LIN {X 262.840,Y 122.534,Z 110.362,A -155.005,B 90.000,C 0.000} C_DIS
LIN {X 263.458,Y 121.203,Z 110.346,A -155.295,B 90.000,C 0.000} C_DIS
LIN {X 263.907,Y 120.222,Z 110.562,A -155.508,B 90.000,C 0.000} C_DIS
LIN {X 264.680,Y 118.510,Z 111.492,A -155.880,B 90.000,C 0.000} C_DIS
LIN {X 264.694,Y 118.479,Z 111.523,A -155.886,B 90.000,C 0.000} C_DIS
LIN {X 264.792,Y 118.258,Z 111.652,A -155.934,B 90.000,C 0.000} C_DIS
LIN {X 265.375,Y 116.944,Z 112.118,A -156.218,B 90.000,C 0.000} C_DIS
LIN {X 265.872,Y 115.810,Z 112.354,A -156.463,B 90.000,C 0.000} C_DIS
LIN {X 265.934,Y 115.668,Z 112.428,A -156.493,B 90.000,C 0.000} C_DIS
LIN {X 266.916,Y 113.380,Z 112.646,A -156.985,B 90.000,C 0.000} C_DIS
LIN {X 267.884,Y 111.074,Z 112.657,A -157.479,B 90.000,C 0.000} C_DIS
LIN {X 268.826,Y 108.776,Z 112.374,A -157.970,B 90.000,C 0.000} C_DIS
LIN {X 268.883,Y 108.638,Z 112.351,A -158.000,B 90.000,C 0.000} C_DIS
LIN {X 269.020,Y 108.296,Z 112.339,A -158.072,B 90.000,C 0.000} C_DIS
LIN {X 268.155,Y 110.420,Z 113.333,A -157.619,B 90.000,C 0.000} C_DIS
LIN {X 267.237,Y 112.623,Z 114.079,A -157.148,B 90.000,C 0.000} C_DIS
LIN {X 266.268,Y 114.897,Z 114.450,A -156.659,B 90.000,C 0.000} C_DIS
LIN {X 266.207,Y 115.038,Z 114.463,A -156.629,B 90.000,C 0.000} C_DIS
LIN {X 265.209,Y 117.321,Z 114.255,A -156.137,B 90.000,C 0.000} C_DIS
LIN {X 264.501,Y 118.908,Z 113.977,A -155.794,B 90.000,C 0.000} C_DIS
LIN {X 264.461,Y 118.998,Z 113.917,A -155.774,B 90.000,C 0.000} C_DIS
LIN {X 264.438,Y 119.048,Z 113.894,A -155.763,B 90.000,C 0.000} C_DIS
LIN {X 263.942,Y 120.144,Z 113.729,A -155.525,B 90.000,C 0.000} C_DIS
LIN {X 263.921,Y 120.190,Z 113.694,A -155.515,B 90.000,C 0.000} C_DIS
LIN {X 263.803,Y 120.449,Z 113.637,A -155.459,B 90.000,C 0.000} C_DIS
LIN {X 263.781,Y 120.497,Z 113.608,A -155.449,B 90.000,C 0.000} C_DIS
LIN {X 263.383,Y 121.365,Z 113.494,A -155.260,B 90.000,C 0.000} C_DIS
LIN {X 263.287,Y 121.574,Z 113.429,A -155.215,B 90.000,C 0.000} C_DIS
LIN {X 262.759,Y 122.709,Z 113.333,A -154.967,B 90.000,C 0.000} C_DIS
LIN {X 262.651,Y 122.941,Z 113.267,A -154.917,B 90.000,C 0.000} C_DIS
LIN {X 262.500,Y 123.263,Z 113.350,A -154.846,B 90.000,C 0.000} C_DIS
LIN {X 262.473,Y 123.319,Z 115.849,A -154.834,B 90.000,C 0.000} C_DIS
LIN {X 262.444,Y 123.381,Z 118.348,A -154.821,B 90.000,C 0.000} C_DIS
LIN {X 262.415,Y 123.444,Z 120.847,A -154.807,B 90.000,C 0.000} C_DIS
LIN {X 262.385,Y 123.507,Z 123.346,A -154.793,B 90.000,C 0.000} C_DIS
LIN {X 262.353,Y 123.575,Z 125.845,A -154.778,B 90.000,C 0.000} C_DIS
LIN {X 262.330,Y 123.623,Z 126.783,A -154.768,B 90.000,C 0.000} C_DIS
LIN {X 262.341,Y 123.600,Z 126.836,A -154.773,B 90.000,C 0.000} C_DIS
LIN {X 262.394,Y 123.488,Z 126.863,A -154.797,B 90.000,C 0.000} C_DIS
LIN {X 262.426,Y 123.421,Z 126.890,A -154.812,B 90.000,C 0.000} C_DIS
LIN {X 262.536,Y 123.186,Z 126.932,A -154.863,B 90.000,C 0.000} C_DIS
LIN {X 263.002,Y 122.188,Z 127.316,A -155.081,B 90.000,C 0.000} C_DIS
LIN {X 263.443,Y 121.234,Z 128.049,A -155.289,B 90.000,C 0.000} C_DIS
LIN {X 263.473,Y 121.169,Z 128.060,A -155.303,B 90.000,C 0.000} C_DIS
LIN {X 263.495,Y 121.122,Z 128.088,A -155.313,B 90.000,C 0.000} C_DIS
LIN {X 263.520,Y 121.068,Z 128.148,A -155.325,B 90.000,C 0.000} C_DIS
LIN {X 263.669,Y 120.742,Z 128.394,A -155.396,B 90.000,C 0.000} C_DIS
LIN {X 263.685,Y 120.708,Z 128.423,A -155.403,B 90.000,C 0.000} C_DIS
LIN {X 263.711,Y 120.649,Z 128.489,A -155.416,B 90.000,C 0.000} C_DIS
LIN {X 263.859,Y 120.325,Z 128.732,A -155.486,B 90.000,C 0.000} C_DIS
LIN {X 263.959,Y 120.107,Z 128.929,A -155.533,B 90.000,C 0.000} C_DIS
LIN {X 264.227,Y 119.517,Z 129.292,A -155.661,B 90.000,C 0.000} C_DIS
LIN {X 264.244,Y 119.478,Z 129.334,A -155.670,B 90.000,C 0.000} C_DIS
LIN {X 264.707,Y 118.449,Z 129.546,A -155.893,B 90.000,C 0.000} C_DIS
LIN {X 264.833,Y 118.167,Z 129.491,A -155.954,B 90.000,C 0.000} C_DIS
LIN {X 264.959,Y 117.884,Z 129.246,A -156.015,B 90.000,C 0.000} C_DIS
LIN {X 265.047,Y 117.686,Z 128.718,A -156.058,B 90.000,C 0.000} C_DIS
LIN {X 265.090,Y 117.589,Z 127.238,A -156.079,B 90.000,C 0.000} C_DIS
LIN {X 265.099,Y 117.569,Z 127.126,A -156.083,B 90.000,C 0.000} C_DIS
LIN {X 265.135,Y 117.488,Z 126.980,A -156.101,B 90.000,C 0.000} C_DIS
LIN {X 265.202,Y 117.336,Z 126.811,A -156.133,B 90.000,C 0.000} C_DIS
LIN {X 265.248,Y 117.232,Z 126.724,A -156.156,B 90.000,C 0.000} C_DIS
LIN {X 265.332,Y 117.043,Z 126.619,A -156.197,B 90.000,C 0.000} C_DIS
LIN {X 265.460,Y 116.751,Z 126.598,A -156.260,B 90.000,C 0.000} C_DIS
LIN {X 265.612,Y 116.405,Z 126.883,A -156.334,B 90.000,C 0.000} C_DIS
LIN {X 265.775,Y 116.033,Z 127.465,A -156.415,B 90.000,C 0.000} C_DIS
LIN {X 265.908,Y 115.728,Z 128.271,A -156.480,B 90.000,C 0.000} C_DIS
LIN {X 266.038,Y 115.429,Z 129.506,A -156.545,B 90.000,C 0.000} C_DIS
RET=EKI_SetBool("oxy","torchState",FALSE)
RET = EKI_Send("oxy","torchState")
PTP {X 264.203,Y 114.633,Z 129.506,A -156.545,B 90.000,C 0.000}
PTP {X 247.690,Y 107.468,Z 129.506,A -156.545,B 90.000,C 0.000}
PTP {X 250.458,Y 100.851,Z 112.225,A -158.067,B 90.000,C 0.000}
PTP {X 267.155,Y 107.574,Z 112.225,A -158.067,B 90.000,C 0.000}
WAIT SEC 2
RET=EKI_SetBool("oxy","torchState",TRUE)
RET = EKI_Send("oxy","torchState")
LIN {X 269.010,Y 108.321,Z 112.225,A -158.067,B 90.000,C 0.000} C_DIS
LIN {X 269.159,Y 107.952,Z 112.154,A -158.146,B 90.000,C 0.000} C_DIS
LIN {X 269.166,Y 107.935,Z 112.107,A -158.149,B 90.000,C 0.000} C_DIS
LIN {X 269.077,Y 108.156,Z 112.139,A -158.102,B 90.000,C 0.000} C_DIS
LIN {X 269.010,Y 108.321,Z 112.225,A -158.067,B 90.000,C 0.000} C_DIS
RET=EKI_SetBool("oxy","torchState",FALSE)
RET = EKI_Send("oxy","torchState")
PTP {X 267.155,Y 107.574,Z 112.225,A -158.067,B 90.000,C 0.000}
PTP {X 250.458,Y 100.851,Z 112.225,A -158.067,B 90.000,C 0.000}
PTP {X 248.222,Y 106.236,Z 107.792,A -156.830,B 90.000,C 0.000}
PTP {X 264.770,Y 113.318,Z 107.792,A -156.830,B 90.000,C 0.000}
WAIT SEC 2
RET=EKI_SetBool("oxy","torchState",TRUE)
RET = EKI_Send("oxy","torchState")
LIN {X 266.608,Y 114.105,Z 107.792,A -156.830,B 90.000,C 0.000} C_DIS
LIN {X 266.579,Y 114.173,Z 107.844,A -156.815,B 90.000,C 0.000} C_DIS
LIN {X 266.518,Y 114.316,Z 107.829,A -156.784,B 90.000,C 0.000} C_DIS
LIN {X 266.499,Y 114.360,Z 107.708,A -156.775,B 90.000,C 0.000} C_DIS
LIN {X 266.520,Y 114.310,Z 107.665,A -156.786,B 90.000,C 0.000} C_DIS
LIN {X 266.543,Y 114.258,Z 107.722,A -156.797,B 90.000,C 0.000} C_DIS
LIN {X 266.582,Y 114.167,Z 107.781,A -156.816,B 90.000,C 0.000} C_DIS
LIN {X 266.608,Y 114.105,Z 107.792,A -156.830,B 90.000,C 0.000} C_DIS
RET=EKI_SetBool("oxy","torchState",FALSE)
RET = EKI_Send("oxy","torchState")
PTP {X 264.770,Y 113.318,Z 107.792,A -156.830,B 90.000,C 0.000}
PTP {X 248.222,Y 106.236,Z 107.792,A -156.830,B 90.000,C 0.000}
PTP {X 248.090,Y 106.544,Z 107.696,A -156.759,B 90.000,C 0.000}
PTP {X 264.629,Y 113.646,Z 107.696,A -156.759,B 90.000,C 0.000}
WAIT SEC 2
RET=EKI_SetBool("oxy","torchState",TRUE)
RET = EKI_Send("oxy","torchState")
LIN {X 266.467,Y 114.436,Z 107.696,A -156.759,B 90.000,C 0.000} C_DIS
LIN {X 266.473,Y 114.420,Z 107.578,A -156.762,B 90.000,C 0.000} C_DIS
LIN {X 266.013,Y 115.486,Z 106.485,A -156.533,B 90.000,C 0.000} C_DIS
LIN {X 265.966,Y 115.593,Z 106.414,A -156.509,B 90.000,C 0.000} C_DIS
LIN {X 265.616,Y 116.396,Z 105.701,A -156.336,B 90.000,C 0.000} C_DIS
LIN {X 265.492,Y 116.679,Z 105.545,A -156.275,B 90.000,C 0.000} C_DIS
LIN {X 265.454,Y 116.766,Z 105.446,A -156.257,B 90.000,C 0.000} C_DIS
LIN {X 265.309,Y 117.094,Z 105.201,A -156.186,B 90.000,C 0.000} C_DIS
LIN {X 265.225,Y 117.284,Z 105.045,A -156.145,B 90.000,C 0.000} C_DIS
LIN {X 265.179,Y 117.388,Z 104.995,A -156.122,B 90.000,C 0.000} C_DIS
LIN {X 265.110,Y 117.544,Z 104.874,A -156.089,B 90.000,C 0.000} C_DIS
LIN {X 265.064,Y 117.648,Z 104.824,A -156.066,B 90.000,C 0.000} C_DIS
LIN {X 265.033,Y 117.718,Z 104.764,A -156.051,B 90.000,C 0.000} C_DIS
LIN {X 264.864,Y 118.098,Z 104.536,A -155.969,B 90.000,C 0.000} C_DIS
LIN {X 264.833,Y 118.168,Z 104.476,A -155.954,B 90.000,C 0.000} C_DIS
LIN {X 264.786,Y 118.271,Z 104.426,A -155.931,B 90.000,C 0.000} C_DIS
LIN {X 264.717,Y 118.427,Z 104.305,A -155.898,B 90.000,C 0.000} C_DIS
LIN {X 264.670,Y 118.531,Z 104.255,A -155.875,B 90.000,C 0.000} C_DIS
LIN {X 264.637,Y 118.605,Z 104.195,A -155.859,B 90.000,C 0.000} C_DIS
LIN {X 264.531,Y 118.843,Z 104.049,A -155.808,B 90.000,C 0.000} C_DIS
LIN {X 264.123,Y 119.746,Z 103.612,A -155.612,B 90.000,C 0.000} C_DIS
LIN {X 264.109,Y 119.776,Z 103.585,A -155.605,B 90.000,C 0.000} C_DIS
LIN {X 263.530,Y 121.045,Z 102.984,A -155.330,B 90.000,C 0.000} C_DIS
LIN {X 262.506,Y 123.250,Z 102.406,A -154.849,B 90.000,C 0.000} C_DIS
LIN {X 261.880,Y 124.575,Z 102.260,A -154.560,B 90.000,C 0.000} C_DIS
LIN {X 261.548,Y 125.270,Z 102.282,A -154.408,B 90.000,C 0.000} C_DIS
LIN {X 261.512,Y 125.345,Z 102.265,A -154.391,B 90.000,C 0.000} C_DIS
LIN {X 260.434,Y 127.569,Z 102.640,A -153.903,B 90.000,C 0.000} C_DIS
LIN {X 259.383,Y 129.695,Z 103.431,A -153.434,B 90.000,C 0.000} C_DIS
LIN {X 258.785,Y 130.883,Z 104.138,A -153.172,B 90.000,C 0.000} C_DIS
LIN {X 258.740,Y 130.971,Z 104.226,A -153.152,B 90.000,C 0.000} C_DIS
LIN {X 258.644,Y 131.162,Z 104.346,A -153.110,B 90.000,C 0.000} C_DIS
LIN {X 258.254,Y 131.927,Z 104.991,A -152.940,B 90.000,C 0.000} C_DIS
LIN {X 258.236,Y 131.963,Z 105.105,A -152.932,B 90.000,C 0.000} C_DIS
LIN {X 257.994,Y 132.436,Z 105.503,A -152.827,B 90.000,C 0.000} C_DIS
LIN {X 257.983,Y 132.457,Z 105.556,A -152.823,B 90.000,C 0.000} C_DIS
LIN {X 257.946,Y 132.530,Z 105.645,A -152.806,B 90.000,C 0.000} C_DIS
LIN {X 257.893,Y 132.632,Z 105.733,A -152.784,B 90.000,C 0.000} C_DIS
LIN {X 257.490,Y 133.413,Z 106.795,A -152.610,B 90.000,C 0.000} C_DIS
LIN {X 257.518,Y 133.358,Z 106.812,A -152.622,B 90.000,C 0.000} C_DIS
LIN {X 258.623,Y 131.196,Z 106.217,A -153.102,B 90.000,C 0.000} C_DIS
LIN {X 259.733,Y 128.992,Z 105.815,A -153.590,B 90.000,C 0.000} C_DIS
LIN {X 260.833,Y 126.752,Z 105.656,A -154.082,B 90.000,C 0.000} C_DIS
LIN {X 260.920,Y 126.573,Z 105.644,A -154.122,B 90.000,C 0.000} C_DIS
LIN {X 260.944,Y 126.524,Z 105.656,A -154.133,B 90.000,C 0.000} C_DIS
LIN {X 262.023,Y 124.272,Z 105.779,A -154.626,B 90.000,C 0.000} C_DIS
LIN {X 262.868,Y 122.477,Z 105.921,A -155.018,B 90.000,C 0.000} C_DIS
LIN {X 263.227,Y 121.703,Z 106.038,A -155.187,B 90.000,C 0.000} C_DIS
LIN {X 263.304,Y 121.535,Z 106.093,A -155.223,B 90.000,C 0.000} C_DIS
LIN {X 263.732,Y 120.604,Z 106.214,A -155.426,B 90.000,C 0.000} C_DIS
LIN {X 263.766,Y 120.530,Z 106.237,A -155.441,B 90.000,C 0.000} C_DIS
LIN {X 263.827,Y 120.397,Z 106.260,A -155.470,B 90.000,C 0.000} C_DIS
LIN {X 263.874,Y 120.294,Z 106.292,A -155.493,B 90.000,C 0.000} C_DIS
LIN {X 263.904,Y 120.227,Z 106.325,A -155.507,B 90.000,C 0.000} C_DIS
LIN {X 264.299,Y 119.357,Z 106.439,A -155.696,B 90.000,C 0.000} C_DIS
LIN {X 264.320,Y 119.310,Z 106.473,A -155.706,B 90.000,C 0.000} C_DIS
LIN {X 264.531,Y 118.843,Z 106.576,A -155.808,B 90.000,C 0.000} C_DIS
LIN {X 264.561,Y 118.776,Z 106.609,A -155.822,B 90.000,C 0.000} C_DIS
LIN {X 265.110,Y 117.545,Z 106.841,A -156.088,B 90.000,C 0.000} C_DIS
LIN {X 265.501,Y 116.659,Z 107.117,A -156.280,B 90.000,C 0.000} C_DIS
LIN {X 265.663,Y 116.290,Z 107.180,A -156.359,B 90.000,C 0.000} C_DIS
LIN {X 265.957,Y 115.616,Z 107.386,A -156.505,B 90.000,C 0.000} C_DIS
LIN {X 265.996,Y 115.525,Z 107.433,A -156.524,B 90.000,C 0.000} C_DIS
LIN {X 266.251,Y 114.938,Z 107.559,A -156.651,B 90.000,C 0.000} C_DIS
LIN {X 266.355,Y 114.695,Z 107.662,A -156.703,B 90.000,C 0.000} C_DIS
LIN {X 266.467,Y 114.436,Z 107.696,A -156.759,B 90.000,C 0.000} C_DIS
RET=EKI_SetBool("oxy","torchState",FALSE)
RET = EKI_Send("oxy","torchState")
PTP {X 264.629,Y 113.646,Z 107.696,A -156.759,B 90.000,C 0.000}
PTP {X 248.090,Y 106.544,Z 107.696,A -156.759,B 90.000,C 0.000}
PTP {X 246.934,Y 109.195,Z 99.474,A -156.145,B 90.000,C 0.000}
PTP {X 263.396,Y 116.475,Z 99.474,A -156.145,B 90.000,C 0.000}
WAIT SEC 2
RET=EKI_SetBool("oxy","torchState",TRUE)
RET = EKI_Send("oxy","torchState")
LIN {X 265.225,Y 117.284,Z 99.474,A -156.145,B 90.000,C 0.000} C_DIS
LIN {X 265.588,Y 116.461,Z 99.674,A -156.322,B 90.000,C 0.000} C_DIS
LIN {X 265.403,Y 116.882,Z 97.216,A -156.232,B 90.000,C 0.000} C_DIS
LIN {X 265.231,Y 117.271,Z 94.753,A -156.148,B 90.000,C 0.000} C_DIS
LIN {X 265.063,Y 117.650,Z 92.288,A -156.066,B 90.000,C 0.000} C_DIS
LIN {X 264.913,Y 117.988,Z 89.815,A -155.993,B 90.000,C 0.000} C_DIS
LIN {X 264.775,Y 118.297,Z 87.338,A -155.926,B 90.000,C 0.000} C_DIS
LIN {X 264.664,Y 118.544,Z 84.853,A -155.872,B 90.000,C 0.000} C_DIS
LIN {X 264.625,Y 118.633,Z 83.669,A -155.853,B 90.000,C 0.000} C_DIS
LIN {X 264.627,Y 118.628,Z 83.485,A -155.854,B 90.000,C 0.000} C_DIS
LIN {X 264.633,Y 118.614,Z 83.419,A -155.857,B 90.000,C 0.000} C_DIS
LIN {X 264.685,Y 118.498,Z 80.922,A -155.882,B 90.000,C 0.000} C_DIS
LIN {X 264.693,Y 118.481,Z 80.815,A -155.886,B 90.000,C 0.000} C_DIS
LIN {X 264.809,Y 118.220,Z 79.843,A -155.942,B 90.000,C 0.000} C_DIS
LIN {X 265.110,Y 117.543,Z 78.071,A -156.089,B 90.000,C 0.000} C_DIS
LIN {X 265.145,Y 117.465,Z 77.909,A -156.106,B 90.000,C 0.000} C_DIS
LIN {X 265.151,Y 117.451,Z 77.852,A -156.109,B 90.000,C 0.000} C_DIS
LIN {X 265.204,Y 117.331,Z 77.610,A -156.135,B 90.000,C 0.000} C_DIS
LIN {X 265.318,Y 117.075,Z 76.873,A -156.190,B 90.000,C 0.000} C_DIS
LIN {X 265.342,Y 117.020,Z 76.771,A -156.202,B 90.000,C 0.000} C_DIS
LIN {X 265.456,Y 116.761,Z 76.088,A -156.258,B 90.000,C 0.000} C_DIS
LIN {X 265.467,Y 116.737,Z 75.974,A -156.263,B 90.000,C 0.000} C_DIS
LIN {X 265.483,Y 116.699,Z 75.860,A -156.271,B 90.000,C 0.000} C_DIS
LIN {X 265.494,Y 116.676,Z 75.823,A -156.276,B 90.000,C 0.000} C_DIS
LIN {X 265.501,Y 116.658,Z 75.717,A -156.280,B 90.000,C 0.000} C_DIS
LIN {X 265.677,Y 116.258,Z 74.324,A -156.366,B 90.000,C 0.000} C_DIS
LIN {X 265.686,Y 116.237,Z 74.139,A -156.371,B 90.000,C 0.000} C_DIS
LIN {X 265.703,Y 116.198,Z 74.040,A -156.379,B 90.000,C 0.000} C_DIS
LIN {X 265.728,Y 116.141,Z 73.812,A -156.392,B 90.000,C 0.000} C_DIS
LIN {X 265.741,Y 116.110,Z 73.758,A -156.398,B 90.000,C 0.000} C_DIS
LIN {X 265.832,Y 115.902,Z 72.391,A -156.443,B 90.000,C 0.000} C_DIS
LIN {X 265.844,Y 115.876,Z 72.304,A -156.449,B 90.000,C 0.000} C_DIS
LIN {X 265.859,Y 115.841,Z 72.048,A -156.456,B 90.000,C 0.000} C_DIS
LIN {X 265.880,Y 115.793,Z 71.864,A -156.466,B 90.000,C 0.000} C_DIS
LIN {X 265.957,Y 115.616,Z 69.371,A -156.505,B 90.000,C 0.000} C_DIS
LIN {X 265.952,Y 115.627,Z 66.871,A -156.502,B 90.000,C 0.000} C_DIS
LIN {X 265.943,Y 115.647,Z 66.003,A -156.498,B 90.000,C 0.000} C_DIS
LIN {X 265.835,Y 115.894,Z 63.518,A -156.445,B 90.000,C 0.000} C_DIS
LIN {X 265.631,Y 116.362,Z 61.071,A -156.344,B 90.000,C 0.000} C_DIS
LIN {X 265.320,Y 117.070,Z 58.693,A -156.191,B 90.000,C 0.000} C_DIS
LIN {X 264.904,Y 118.007,Z 56.413,A -155.988,B 90.000,C 0.000} C_DIS
LIN {X 264.399,Y 119.136,Z 54.241,A -155.744,B 90.000,C 0.000} C_DIS
LIN {X 264.143,Y 119.702,Z 53.360,A -155.621,B 90.000,C 0.000} C_DIS
LIN {X 264.062,Y 119.879,Z 53.046,A -155.583,B 90.000,C 0.000} C_DIS
LIN {X 263.992,Y 120.035,Z 52.849,A -155.549,B 90.000,C 0.000} C_DIS
LIN {X 263.519,Y 121.070,Z 51.308,A -155.324,B 90.000,C 0.000} C_DIS
LIN {X 263.497,Y 121.118,Z 51.250,A -155.314,B 90.000,C 0.000} C_DIS
LIN {X 263.460,Y 121.197,Z 51.174,A -155.297,B 90.000,C 0.000} C_DIS
LIN {X 263.376,Y 121.380,Z 50.910,A -155.257,B 90.000,C 0.000} C_DIS
LIN {X 263.352,Y 121.432,Z 50.855,A -155.246,B 90.000,C 0.000} C_DIS
LIN {X 263.328,Y 121.483,Z 50.838,A -155.234,B 90.000,C 0.000} C_DIS
LIN {X 263.161,Y 121.845,Z 50.307,A -155.156,B 90.000,C 0.000} C_DIS
LIN {X 263.113,Y 121.948,Z 50.265,A -155.133,B 90.000,C 0.000} C_DIS
LIN {X 262.946,Y 122.309,Z 49.734,A -155.054,B 90.000,C 0.000} C_DIS
LIN {X 262.922,Y 122.361,Z 49.717,A -155.043,B 90.000,C 0.000} C_DIS
LIN {X 262.898,Y 122.412,Z 49.693,A -155.032,B 90.000,C 0.000} C_DIS
LIN {X 262.439,Y 123.393,Z 48.607,A -154.818,B 90.000,C 0.000} C_DIS
LIN {X 262.392,Y 123.492,Z 48.437,A -154.796,B 90.000,C 0.000} C_DIS
LIN {X 262.197,Y 123.906,Z 47.963,A -154.706,B 90.000,C 0.000} C_DIS
LIN {X 261.367,Y 125.648,Z 46.374,A -154.325,B 90.000,C 0.000} C_DIS
LIN {X 261.351,Y 125.681,Z 46.344,A -154.318,B 90.000,C 0.000} C_DIS
LIN {X 261.351,Y 125.681,Z 46.344,A -154.318,B 90.000,C 0.000} C_DIS
LIN {X 261.334,Y 125.717,Z 46.279,A -154.310,B 90.000,C 0.000} C_DIS
LIN {X 261.321,Y 125.742,Z 46.355,A -154.304,B 90.000,C 0.000} C_DIS
LIN {X 261.350,Y 125.683,Z 46.514,A -154.317,B 90.000,C 0.000} C_DIS
LIN {X 261.389,Y 125.601,Z 46.639,A -154.335,B 90.000,C 0.000} C_DIS
LIN {X 261.870,Y 124.596,Z 48.877,A -154.555,B 90.000,C 0.000} C_DIS
LIN {X 262.236,Y 123.824,Z 51.226,A -154.724,B 90.000,C 0.000} C_DIS
LIN {X 262.491,Y 123.283,Z 53.653,A -154.842,B 90.000,C 0.000} C_DIS
LIN {X 262.662,Y 122.918,Z 56.121,A -154.922,B 90.000,C 0.000} C_DIS
LIN {X 262.755,Y 122.719,Z 58.611,A -154.965,B 90.000,C 0.000} C_DIS
LIN {X 262.814,Y 122.593,Z 59.986,A -154.993,B 90.000,C 0.000} C_DIS
LIN {X 262.790,Y 122.644,Z 60.102,A -154.982,B 90.000,C 0.000} C_DIS
LIN {X 262.861,Y 122.492,Z 62.142,A -155.015,B 90.000,C 0.000} C_DIS
LIN {X 262.853,Y 122.508,Z 62.263,A -155.011,B 90.000,C 0.000} C_DIS
LIN {X 262.873,Y 122.466,Z 63.107,A -155.020,B 90.000,C 0.000} C_DIS
LIN {X 262.869,Y 122.473,Z 63.287,A -155.019,B 90.000,C 0.000} C_DIS
LIN {X 262.862,Y 122.490,Z 63.386,A -155.015,B 90.000,C 0.000} C_DIS
LIN {X 262.909,Y 122.388,Z 65.674,A -155.037,B 90.000,C 0.000} C_DIS
LIN {X 262.905,Y 122.396,Z 65.733,A -155.036,B 90.000,C 0.000} C_DIS
LIN {X 262.909,Y 122.389,Z 66.516,A -155.037,B 90.000,C 0.000} C_DIS
LIN {X 262.900,Y 122.407,Z 66.587,A -155.033,B 90.000,C 0.000} C_DIS
LIN {X 262.890,Y 122.430,Z 69.087,A -155.028,B 90.000,C 0.000} C_DIS
LIN {X 262.846,Y 122.523,Z 71.584,A -155.008,B 90.000,C 0.000} C_DIS
LIN {X 262.768,Y 122.691,Z 73.940,A -154.971,B 90.000,C 0.000} C_DIS
LIN {X 262.745,Y 122.741,Z 74.097,A -154.960,B 90.000,C 0.000} C_DIS
LIN {X 262.566,Y 123.123,Z 76.561,A -154.877,B 90.000,C 0.000} C_DIS
LIN {X 262.392,Y 123.492,Z 77.966,A -154.797,B 90.000,C 0.000} C_DIS
LIN {X 262.239,Y 123.817,Z 78.614,A -154.725,B 90.000,C 0.000} C_DIS
LIN {X 262.197,Y 123.906,Z 78.734,A -154.706,B 90.000,C 0.000} C_DIS
LIN {X 262.124,Y 124.060,Z 78.900,A -154.672,B 90.000,C 0.000} C_DIS
LIN {X 261.990,Y 124.343,Z 79.104,A -154.611,B 90.000,C 0.000} C_DIS
LIN {X 261.942,Y 124.443,Z 79.194,A -154.589,B 90.000,C 0.000} C_DIS
LIN {X 261.786,Y 124.772,Z 79.226,A -154.517,B 90.000,C 0.000} C_DIS
LIN {X 261.534,Y 125.300,Z 79.049,A -154.401,B 90.000,C 0.000} C_DIS
LIN {X 261.270,Y 125.849,Z 78.581,A -154.281,B 90.000,C 0.000} C_DIS
LIN {X 260.993,Y 126.422,Z 77.795,A -154.155,B 90.000,C 0.000} C_DIS
LIN {X 260.897,Y 126.621,Z 77.365,A -154.111,B 90.000,C 0.000} C_DIS
LIN {X 260.603,Y 127.225,Z 74.957,A -153.979,B 90.000,C 0.000} C_DIS
LIN {X 260.574,Y 127.283,Z 74.674,A -153.966,B 90.000,C 0.000} C_DIS
LIN {X 260.530,Y 127.374,Z 73.722,A -153.946,B 90.000,C 0.000} C_DIS
LIN {X 260.523,Y 127.387,Z 71.222,A -153.943,B 90.000,C 0.000} C_DIS
LIN {X 260.521,Y 127.393,Z 70.171,A -153.942,B 90.000,C 0.000} C_DIS
LIN {X 260.609,Y 127.213,Z 67.679,A -153.981,B 90.000,C 0.000} C_DIS
LIN {X 260.664,Y 127.100,Z 66.644,A -154.006,B 90.000,C 0.000} C_DIS
LIN {X 260.686,Y 127.053,Z 66.459,A -154.016,B 90.000,C 0.000} C_DIS
LIN {X 260.792,Y 126.836,Z 64.752,A -154.064,B 90.000,C 0.000} C_DIS
LIN {X 260.798,Y 126.825,Z 64.553,A -154.067,B 90.000,C 0.000} C_DIS
LIN {X 260.881,Y 126.653,Z 63.397,A -154.104,B 90.000,C 0.000} C_DIS
LIN {X 260.915,Y 126.583,Z 63.244,A -154.120,B 90.000,C 0.000} C_DIS
LIN {X 260.929,Y 126.555,Z 63.068,A -154.126,B 90.000,C 0.000} C_DIS
LIN {X 260.921,Y 126.570,Z 62.922,A -154.122,B 90.000,C 0.000} C_DIS
LIN {X 260.862,Y 126.693,Z 62.949,A -154.095,B 90.000,C 0.000} C_DIS
LIN {X 260.789,Y 126.843,Z 63.075,A -154.062,B 90.000,C 0.000} C_DIS
LIN {X 260.719,Y 126.986,Z 63.230,A -154.031,B 90.000,C 0.000} C_DIS
LIN {X 260.522,Y 127.391,Z 63.571,A -153.942,B 90.000,C 0.000} C_DIS
LIN {X 260.464,Y 127.508,Z 63.744,A -153.916,B 90.000,C 0.000} C_DIS
LIN {X 260.245,Y 127.955,Z 64.147,A -153.818,B 90.000,C 0.000} C_DIS
LIN {X 260.009,Y 128.435,Z 64.781,A -153.712,B 90.000,C 0.000} C_DIS
LIN {X 259.970,Y 128.513,Z 64.850,A -153.695,B 90.000,C 0.000} C_DIS
LIN {X 259.932,Y 128.591,Z 64.941,A -153.678,B 90.000,C 0.000} C_DIS
LIN {X 259.919,Y 128.615,Z 64.994,A -153.673,B 90.000,C 0.000} C_DIS
LIN {X 259.893,Y 128.669,Z 65.049,A -153.661,B 90.000,C 0.000} C_DIS
LIN {X 259.589,Y 129.281,Z 65.893,A -153.526,B 90.000,C 0.000} C_DIS
LIN {X 259.528,Y 129.403,Z 66.141,A -153.499,B 90.000,C 0.000} C_DIS
LIN {X 259.507,Y 129.446,Z 66.269,A -153.489,B 90.000,C 0.000} C_DIS
LIN {X 259.492,Y 129.476,Z 66.302,A -153.483,B 90.000,C 0.000} C_DIS
LIN {X 259.360,Y 129.739,Z 66.751,A -153.425,B 90.000,C 0.000} C_DIS
LIN {X 259.341,Y 129.778,Z 66.881,A -153.416,B 90.000,C 0.000} C_DIS
LIN {X 259.127,Y 130.204,Z 67.725,A -153.322,B 90.000,C 0.000} C_DIS
LIN {X 259.030,Y 130.397,Z 68.237,A -153.279,B 90.000,C 0.000} C_DIS
LIN {X 259.022,Y 130.413,Z 68.359,A -153.276,B 90.000,C 0.000} C_DIS
LIN {X 259.026,Y 130.405,Z 68.445,A -153.277,B 90.000,C 0.000} C_DIS
LIN {X 258.980,Y 130.497,Z 68.426,A -153.257,B 90.000,C 0.000} C_DIS
LIN {X 258.983,Y 130.490,Z 68.510,A -153.259,B 90.000,C 0.000} C_DIS
LIN {X 258.974,Y 130.508,Z 68.647,A -153.254,B 90.000,C 0.000} C_DIS
LIN {X 258.915,Y 130.625,Z 69.141,A -153.229,B 90.000,C 0.000} C_DIS
LIN {X 258.906,Y 130.643,Z 69.375,A -153.225,B 90.000,C 0.000} C_DIS
LIN {X 258.849,Y 130.756,Z 69.877,A -153.200,B 90.000,C 0.000} C_DIS
LIN {X 258.836,Y 130.782,Z 69.942,A -153.194,B 90.000,C 0.000} C_DIS
LIN {X 258.735,Y 130.982,Z 71.312,A -153.150,B 90.000,C 0.000} C_DIS
LIN {X 258.719,Y 131.012,Z 71.366,A -153.143,B 90.000,C 0.000} C_DIS
LIN {X 258.703,Y 131.046,Z 71.480,A -153.136,B 90.000,C 0.000} C_DIS
LIN {X 258.679,Y 131.092,Z 71.878,A -153.125,B 90.000,C 0.000} C_DIS
LIN {X 258.653,Y 131.143,Z 72.034,A -153.114,B 90.000,C 0.000} C_DIS
LIN {X 258.583,Y 131.282,Z 73.457,A -153.083,B 90.000,C 0.000} C_DIS
LIN {X 258.566,Y 131.316,Z 73.585,A -153.076,B 90.000,C 0.000} C_DIS
LIN {X 258.551,Y 131.345,Z 73.770,A -153.069,B 90.000,C 0.000} C_DIS
LIN {X 258.523,Y 131.400,Z 76.269,A -153.057,B 90.000,C 0.000} C_DIS
LIN {X 258.517,Y 131.411,Z 77.392,A -153.055,B 90.000,C 0.000} C_DIS
LIN {X 258.710,Y 131.032,Z 79.855,A -153.139,B 90.000,C 0.000} C_DIS
LIN {X 258.772,Y 130.908,Z 80.389,A -153.166,B 90.000,C 0.000} C_DIS
LIN {X 258.794,Y 130.865,Z 80.389,A -153.176,B 90.000,C 0.000} C_DIS
LIN {X 259.029,Y 130.400,Z 81.436,A -153.279,B 90.000,C 0.000} C_DIS
LIN {X 259.127,Y 130.204,Z 81.774,A -153.322,B 90.000,C 0.000} C_DIS
LIN {X 259.207,Y 130.044,Z 82.001,A -153.357,B 90.000,C 0.000} C_DIS
LIN {X 259.477,Y 129.505,Z 82.616,A -153.476,B 90.000,C 0.000} C_DIS
LIN {X 259.716,Y 129.026,Z 82.973,A -153.582,B 90.000,C 0.000} C_DIS
LIN {X 259.817,Y 128.822,Z 83.033,A -153.627,B 90.000,C 0.000} C_DIS
LIN {X 259.850,Y 128.755,Z 83.086,A -153.642,B 90.000,C 0.000} C_DIS
LIN {X 259.882,Y 128.691,Z 83.541,A -153.656,B 90.000,C 0.000} C_DIS
LIN {X 259.828,Y 128.799,Z 86.038,A -153.632,B 90.000,C 0.000} C_DIS
LIN {X 259.785,Y 128.886,Z 88.536,A -153.613,B 90.000,C 0.000} C_DIS
LIN {X 259.752,Y 128.953,Z 91.035,A -153.598,B 90.000,C 0.000} C_DIS
LIN {X 259.731,Y 128.995,Z 93.535,A -153.589,B 90.000,C 0.000} C_DIS
LIN {X 259.699,Y 129.059,Z 95.774,A -153.575,B 90.000,C 0.000} C_DIS
LIN {X 259.617,Y 129.225,Z 96.400,A -153.538,B 90.000,C 0.000} C_DIS
LIN {X 259.485,Y 129.489,Z 97.083,A -153.480,B 90.000,C 0.000} C_DIS
LIN {X 259.407,Y 129.646,Z 97.367,A -153.445,B 90.000,C 0.000} C_DIS
LIN {X 259.387,Y 129.685,Z 97.481,A -153.436,B 90.000,C 0.000} C_DIS
LIN {X 259.331,Y 129.798,Z 97.652,A -153.411,B 90.000,C 0.000} C_DIS
LIN {X 259.316,Y 129.828,Z 97.685,A -153.405,B 90.000,C 0.000} C_DIS
LIN {X 259.043,Y 130.372,Z 98.512,A -153.285,B 90.000,C 0.000} C_DIS
LIN {X 259.031,Y 130.396,Z 98.617,A -153.279,B 90.000,C 0.000} C_DIS
LIN {X 259.403,Y 129.653,Z 98.473,A -153.444,B 90.000,C 0.000} C_DIS
LIN {X 260.503,Y 127.425,Z 98.198,A -153.934,B 90.000,C 0.000} C_DIS
LIN {X 261.593,Y 125.176,Z 98.161,A -154.428,B 90.000,C 0.000} C_DIS
LIN {X 262.660,Y 122.921,Z 98.330,A -154.921,B 90.000,C 0.000} C_DIS
LIN {X 262.988,Y 122.219,Z 98.412,A -155.074,B 90.000,C 0.000} C_DIS
LIN {X 263.042,Y 122.103,Z 98.469,A -155.099,B 90.000,C 0.000} C_DIS
LIN {X 263.508,Y 121.093,Z 98.581,A -155.319,B 90.000,C 0.000} C_DIS
LIN {X 263.589,Y 120.916,Z 98.649,A -155.358,B 90.000,C 0.000} C_DIS
LIN {X 264.199,Y 119.579,Z 98.877,A -155.648,B 90.000,C 0.000} C_DIS
LIN {X 265.192,Y 117.359,Z 99.455,A -156.129,B 90.000,C 0.000} C_DIS
LIN {X 265.225,Y 117.284,Z 99.474,A -156.145,B 90.000,C 0.000} C_DIS
RET=EKI_SetBool("oxy","torchState",FALSE)
RET = EKI_Send("oxy","torchState")
PTP {X 263.396,Y 116.475,Z 99.474,A -156.145,B 90.000,C 0.000}
PTP {X 246.934,Y 109.195,Z 99.474,A -156.145,B 90.000,C 0.000}
PTP {X 240.690,Y 122.345,Z 121.667,A -153.055,B 90.000,C 0.000}
PTP {X 256.736,Y 130.501,Z 121.667,A -153.055,B 90.000,C 0.000}
WAIT SEC 2
RET=EKI_SetBool("oxy","torchState",TRUE)
RET = EKI_Send("oxy","torchState")
LIN {X 258.519,Y 131.407,Z 121.667,A -153.055,B 90.000,C 0.000} C_DIS
LIN {X 258.587,Y 131.274,Z 121.574,A -153.085,B 90.000,C 0.000} C_DIS
LIN {X 257.448,Y 133.494,Z 121.429,A -152.592,B 90.000,C 0.000} C_DIS
LIN {X 256.642,Y 135.037,Z 121.247,A -152.248,B 90.000,C 0.000} C_DIS
LIN {X 256.558,Y 135.195,Z 121.187,A -152.213,B 90.000,C 0.000} C_DIS
LIN {X 256.127,Y 136.011,Z 121.065,A -152.030,B 90.000,C 0.000} C_DIS
LIN {X 256.089,Y 136.082,Z 121.042,A -152.015,B 90.000,C 0.000} C_DIS
LIN {X 256.021,Y 136.211,Z 121.020,A -151.986,B 90.000,C 0.000} C_DIS
LIN {X 255.967,Y 136.311,Z 120.982,A -151.963,B 90.000,C 0.000} C_DIS
LIN {X 255.941,Y 136.361,Z 120.951,A -151.952,B 90.000,C 0.000} C_DIS
LIN {X 254.998,Y 138.116,Z 120.466,A -151.559,B 90.000,C 0.000} C_DIS
LIN {X 254.944,Y 138.216,Z 120.451,A -151.536,B 90.000,C 0.000} C_DIS
LIN {X 254.835,Y 138.417,Z 120.382,A -151.491,B 90.000,C 0.000} C_DIS
LIN {X 254.798,Y 138.484,Z 120.341,A -151.476,B 90.000,C 0.000} C_DIS
LIN {X 254.758,Y 138.558,Z 120.310,A -151.459,B 90.000,C 0.000} C_DIS
LIN {X 254.700,Y 138.666,Z 120.302,A -151.435,B 90.000,C 0.000} C_DIS
LIN {X 254.284,Y 139.427,Z 120.000,A -151.263,B 90.000,C 0.000} C_DIS
LIN {X 254.263,Y 139.464,Z 119.948,A -151.255,B 90.000,C 0.000} C_DIS
LIN {X 254.208,Y 139.564,Z 119.915,A -151.233,B 90.000,C 0.000} C_DIS
LIN {X 254.154,Y 139.664,Z 119.904,A -151.210,B 90.000,C 0.000} C_DIS
LIN {X 253.438,Y 140.958,Z 119.213,A -150.918,B 90.000,C 0.000} C_DIS
LIN {X 253.404,Y 141.019,Z 119.158,A -150.904,B 90.000,C 0.000} C_DIS
LIN {X 252.604,Y 142.448,Z 118.175,A -150.581,B 90.000,C 0.000} C_DIS
LIN {X 252.419,Y 142.775,Z 117.866,A -150.506,B 90.000,C 0.000} C_DIS
LIN {X 252.346,Y 142.905,Z 117.768,A -150.477,B 90.000,C 0.000} C_DIS
LIN {X 251.846,Y 143.784,Z 116.881,A -150.277,B 90.000,C 0.000} C_DIS
LIN {X 251.365,Y 144.623,Z 115.672,A -150.086,B 90.000,C 0.000} C_DIS
LIN {X 250.892,Y 145.441,Z 113.921,A -149.899,B 90.000,C 0.000} C_DIS
LIN {X 250.579,Y 145.981,Z 111.559,A -149.776,B 90.000,C 0.000} C_DIS
LIN {X 250.560,Y 146.013,Z 111.025,A -149.769,B 90.000,C 0.000} C_DIS
LIN {X 250.662,Y 145.837,Z 108.534,A -149.809,B 90.000,C 0.000} C_DIS
LIN {X 250.665,Y 145.832,Z 108.458,A -149.810,B 90.000,C 0.000} C_DIS
LIN {X 250.683,Y 145.802,Z 108.405,A -149.817,B 90.000,C 0.000} C_DIS
LIN {X 250.701,Y 145.770,Z 108.291,A -149.824,B 90.000,C 0.000} C_DIS
LIN {X 250.806,Y 145.589,Z 107.444,A -149.866,B 90.000,C 0.000} C_DIS
LIN {X 250.825,Y 145.557,Z 107.267,A -149.873,B 90.000,C 0.000} C_DIS
LIN {X 250.974,Y 145.300,Z 106.471,A -149.932,B 90.000,C 0.000} C_DIS
LIN {X 250.990,Y 145.272,Z 106.357,A -149.938,B 90.000,C 0.000} C_DIS
LIN {X 251.081,Y 145.115,Z 106.072,A -149.974,B 90.000,C 0.000} C_DIS
LIN {X 251.109,Y 145.067,Z 106.005,A -149.985,B 90.000,C 0.000} C_DIS
LIN {X 251.518,Y 144.357,Z 104.705,A -150.147,B 90.000,C 0.000} C_DIS
LIN {X 251.906,Y 143.678,Z 104.010,A -150.301,B 90.000,C 0.000} C_DIS
LIN {X 251.993,Y 143.526,Z 103.910,A -150.336,B 90.000,C 0.000} C_DIS
LIN {X 252.002,Y 143.509,Z 103.858,A -150.339,B 90.000,C 0.000} C_DIS
LIN {X 252.417,Y 142.778,Z 103.352,A -150.506,B 90.000,C 0.000} C_DIS
LIN {X 252.454,Y 142.713,Z 100.853,A -150.520,B 90.000,C 0.000} C_DIS
LIN {X 252.493,Y 142.644,Z 98.355,A -150.536,B 90.000,C 0.000} C_DIS
LIN {X 252.525,Y 142.587,Z 95.855,A -150.549,B 90.000,C 0.000} C_DIS
LIN {X 252.560,Y 142.525,Z 93.357,A -150.563,B 90.000,C 0.000} C_DIS
LIN {X 252.594,Y 142.465,Z 90.858,A -150.577,B 90.000,C 0.000} C_DIS
LIN {X 252.631,Y 142.400,Z 89.264,A -150.591,B 90.000,C 0.000} C_DIS
LIN {X 252.777,Y 142.140,Z 88.807,A -150.650,B 90.000,C 0.000} C_DIS
LIN {X 252.827,Y 142.051,Z 88.715,A -150.671,B 90.000,C 0.000} C_DIS
LIN {X 253.278,Y 141.245,Z 87.467,A -150.853,B 90.000,C 0.000} C_DIS
LIN {X 253.299,Y 141.207,Z 87.382,A -150.862,B 90.000,C 0.000} C_DIS
LIN {X 253.329,Y 141.154,Z 87.297,A -150.874,B 90.000,C 0.000} C_DIS
LIN {X 253.351,Y 141.115,Z 87.183,A -150.883,B 90.000,C 0.000} C_DIS
LIN {X 253.441,Y 140.953,Z 86.970,A -150.919,B 90.000,C 0.000} C_DIS
LIN {X 253.522,Y 140.806,Z 86.728,A -150.952,B 90.000,C 0.000} C_DIS
LIN {X 253.560,Y 140.738,Z 86.571,A -150.968,B 90.000,C 0.000} C_DIS
LIN {X 253.607,Y 140.654,Z 86.443,A -150.987,B 90.000,C 0.000} C_DIS
LIN {X 253.660,Y 140.558,Z 86.225,A -151.008,B 90.000,C 0.000} C_DIS
LIN {X 253.718,Y 140.453,Z 86.060,A -151.032,B 90.000,C 0.000} C_DIS
LIN {X 253.824,Y 140.262,Z 85.689,A -151.075,B 90.000,C 0.000} C_DIS
LIN {X 254.153,Y 139.664,Z 84.419,A -151.210,B 90.000,C 0.000} C_DIS
LIN {X 254.181,Y 139.614,Z 84.338,A -151.221,B 90.000,C 0.000} C_DIS
LIN {X 254.204,Y 139.572,Z 84.295,A -151.231,B 90.000,C 0.000} C_DIS
LIN {X 254.263,Y 139.464,Z 83.884,A -151.255,B 90.000,C 0.000} C_DIS
LIN {X 254.284,Y 139.427,Z 83.817,A -151.263,B 90.000,C 0.000} C_DIS
LIN {X 254.513,Y 139.007,Z 82.859,A -151.358,B 90.000,C 0.000} C_DIS
LIN {X 254.531,Y 138.974,Z 82.745,A -151.365,B 90.000,C 0.000} C_DIS
LIN {X 254.646,Y 138.765,Z 82.204,A -151.413,B 90.000,C 0.000} C_DIS
LIN {X 254.798,Y 138.484,Z 81.406,A -151.476,B 90.000,C 0.000} C_DIS
LIN {X 254.806,Y 138.471,Z 81.323,A -151.479,B 90.000,C 0.000} C_DIS
LIN {X 254.946,Y 138.213,Z 80.609,A -151.537,B 90.000,C 0.000} C_DIS
LIN {X 255.192,Y 137.757,Z 78.862,A -151.639,B 90.000,C 0.000} C_DIS
LIN {X 255.218,Y 137.709,Z 78.819,A -151.650,B 90.000,C 0.000} C_DIS
LIN {X 255.234,Y 137.680,Z 78.705,A -151.656,B 90.000,C 0.000} C_DIS
LIN {X 255.264,Y 137.623,Z 78.307,A -151.669,B 90.000,C 0.000} C_DIS
LIN {X 255.360,Y 137.446,Z 77.681,A -151.709,B 90.000,C 0.000} C_DIS
LIN {X 255.384,Y 137.400,Z 77.283,A -151.719,B 90.000,C 0.000} C_DIS
LIN {X 255.427,Y 137.322,Z 76.942,A -151.737,B 90.000,C 0.000} C_DIS
LIN {X 255.442,Y 137.292,Z 76.868,A -151.743,B 90.000,C 0.000} C_DIS
LIN {X 255.616,Y 136.969,Z 74.495,A -151.816,B 90.000,C 0.000} C_DIS
LIN {X 255.638,Y 136.928,Z 74.339,A -151.825,B 90.000,C 0.000} C_DIS
LIN {X 255.692,Y 136.827,Z 71.841,A -151.848,B 90.000,C 0.000} C_DIS
LIN {X 255.704,Y 136.804,Z 69.374,A -151.853,B 90.000,C 0.000} C_DIS
LIN {X 255.712,Y 136.790,Z 69.313,A -151.856,B 90.000,C 0.000} C_DIS
LIN {X 255.580,Y 137.036,Z 66.829,A -151.801,B 90.000,C 0.000} C_DIS
LIN {X 255.354,Y 137.457,Z 64.375,A -151.706,B 90.000,C 0.000} C_DIS
LIN {X 255.046,Y 138.028,Z 61.961,A -151.578,B 90.000,C 0.000} C_DIS
LIN {X 254.663,Y 138.732,Z 59.593,A -151.420,B 90.000,C 0.000} C_DIS
LIN {X 254.300,Y 139.396,Z 57.796,A -151.270,B 90.000,C 0.000} C_DIS
LIN {X 254.300,Y 139.396,Z 57.796,A -151.270,B 90.000,C 0.000} C_DIS
LIN {X 254.206,Y 139.569,Z 57.483,A -151.232,B 90.000,C 0.000} C_DIS
LIN {X 254.171,Y 139.632,Z 57.534,A -151.217,B 90.000,C 0.000} C_DIS
LIN {X 254.288,Y 139.419,Z 60.022,A -151.265,B 90.000,C 0.000} C_DIS
LIN {X 254.353,Y 139.300,Z 62.518,A -151.292,B 90.000,C 0.000} C_DIS
LIN {X 254.358,Y 139.291,Z 62.657,A -151.294,B 90.000,C 0.000} C_DIS
LIN {X 254.350,Y 139.305,Z 62.718,A -151.291,B 90.000,C 0.000} C_DIS
LIN {X 254.323,Y 139.356,Z 65.217,A -151.280,B 90.000,C 0.000} C_DIS
LIN {X 254.250,Y 139.488,Z 67.712,A -151.250,B 90.000,C 0.000} C_DIS
LIN {X 254.236,Y 139.514,Z 68.066,A -151.244,B 90.000,C 0.000} C_DIS
LIN {X 254.219,Y 139.545,Z 68.194,A -151.237,B 90.000,C 0.000} C_DIS
LIN {X 254.057,Y 139.839,Z 70.671,A -151.171,B 90.000,C 0.000} C_DIS
LIN {X 253.820,Y 140.270,Z 73.122,A -151.073,B 90.000,C 0.000} C_DIS
LIN {X 253.756,Y 140.385,Z 73.814,A -151.047,B 90.000,C 0.000} C_DIS
LIN {X 253.440,Y 140.955,Z 75.917,A -150.919,B 90.000,C 0.000} C_DIS
LIN {X 253.284,Y 141.234,Z 76.767,A -150.856,B 90.000,C 0.000} C_DIS
LIN {X 253.279,Y 141.244,Z 76.847,A -150.853,B 90.000,C 0.000} C_DIS
LIN {X 253.124,Y 141.520,Z 77.624,A -150.791,B 90.000,C 0.000} C_DIS
LIN {X 253.119,Y 141.530,Z 77.681,A -150.789,B 90.000,C 0.000} C_DIS
LIN {X 253.110,Y 141.546,Z 77.738,A -150.785,B 90.000,C 0.000} C_DIS
LIN {X 252.994,Y 141.754,Z 78.279,A -150.738,B 90.000,C 0.000} C_DIS
LIN {X 252.973,Y 141.790,Z 78.421,A -150.730,B 90.000,C 0.000} C_DIS
LIN {X 252.656,Y 142.355,Z 79.673,A -150.602,B 90.000,C 0.000} C_DIS
LIN {X 252.565,Y 142.516,Z 80.128,A -150.565,B 90.000,C 0.000} C_DIS
LIN {X 252.536,Y 142.568,Z 80.217,A -150.553,B 90.000,C 0.000} C_DIS
LIN {X 252.492,Y 142.646,Z 80.388,A -150.536,B 90.000,C 0.000} C_DIS
LIN {X 252.462,Y 142.698,Z 80.469,A -150.524,B 90.000,C 0.000} C_DIS
LIN {X 252.438,Y 142.742,Z 80.583,A -150.514,B 90.000,C 0.000} C_DIS
LIN {X 252.378,Y 142.847,Z 80.754,A -150.490,B 90.000,C 0.000} C_DIS
LIN {X 252.354,Y 142.890,Z 80.867,A -150.480,B 90.000,C 0.000} C_DIS
LIN {X 252.307,Y 142.972,Z 81.010,A -150.462,B 90.000,C 0.000} C_DIS
LIN {X 252.271,Y 143.036,Z 81.152,A -150.447,B 90.000,C 0.000} C_DIS
LIN {X 252.091,Y 143.353,Z 81.607,A -150.375,B 90.000,C 0.000} C_DIS
LIN {X 252.082,Y 143.368,Z 81.655,A -150.372,B 90.000,C 0.000} C_DIS
LIN {X 252.007,Y 143.501,Z 81.971,A -150.341,B 90.000,C 0.000} C_DIS
LIN {X 251.911,Y 143.669,Z 82.213,A -150.303,B 90.000,C 0.000} C_DIS
LIN {X 251.789,Y 143.883,Z 82.572,A -150.255,B 90.000,C 0.000} C_DIS
LIN {X 251.740,Y 143.969,Z 82.664,A -150.235,B 90.000,C 0.000} C_DIS
LIN {X 251.558,Y 144.286,Z 83.222,A -150.163,B 90.000,C 0.000} C_DIS
LIN {X 250.720,Y 145.737,Z 85.077,A -149.832,B 90.000,C 0.000} C_DIS
LIN {X 249.997,Y 146.974,Z 86.386,A -149.549,B 90.000,C 0.000} C_DIS
LIN {X 249.718,Y 147.447,Z 86.959,A -149.440,B 90.000,C 0.000} C_DIS
LIN {X 249.709,Y 147.464,Z 87.012,A -149.436,B 90.000,C 0.000} C_DIS
LIN {X 249.400,Y 147.986,Z 87.585,A -149.316,B 90.000,C 0.000} C_DIS
LIN {X 249.386,Y 148.010,Z 87.638,A -149.311,B 90.000,C 0.000} C_DIS
LIN {X 249.355,Y 148.061,Z 87.698,A -149.299,B 90.000,C 0.000} C_DIS
LIN {X 248.809,Y 148.977,Z 89.091,A -149.088,B 90.000,C 0.000} C_DIS
LIN {X 248.760,Y 149.059,Z 89.241,A -149.070,B 90.000,C 0.000} C_DIS
LIN {X 248.735,Y 149.100,Z 89.369,A -149.060,B 90.000,C 0.000} C_DIS
LIN {X 248.718,Y 149.128,Z 89.402,A -149.054,B 90.000,C 0.000} C_DIS
LIN {X 248.653,Y 149.237,Z 89.573,A -149.029,B 90.000,C 0.000} C_DIS
LIN {X 248.631,Y 149.274,Z 89.686,A -149.020,B 90.000,C 0.000} C_DIS
LIN {X 248.508,Y 149.478,Z 90.052,A -148.973,B 90.000,C 0.000} C_DIS
LIN {X 248.433,Y 149.603,Z 90.312,A -148.944,B 90.000,C 0.000} C_DIS
LIN {X 248.206,Y 149.979,Z 91.300,A -148.857,B 90.000,C 0.000} C_DIS
LIN {X 248.156,Y 150.062,Z 91.418,A -148.838,B 90.000,C 0.000} C_DIS
LIN {X 247.941,Y 150.417,Z 92.304,A -148.756,B 90.000,C 0.000} C_DIS
LIN {X 247.921,Y 150.450,Z 92.531,A -148.749,B 90.000,C 0.000} C_DIS
LIN {X 247.801,Y 150.647,Z 93.072,A -148.703,B 90.000,C 0.000} C_DIS
LIN {X 247.788,Y 150.668,Z 93.161,A -148.698,B 90.000,C 0.000} C_DIS
LIN {X 247.771,Y 150.698,Z 93.214,A -148.691,B 90.000,C 0.000} C_DIS
LIN {X 247.751,Y 150.729,Z 93.328,A -148.684,B 90.000,C 0.000} C_DIS
LIN {X 247.744,Y 150.740,Z 93.441,A -148.682,B 90.000,C 0.000} C_DIS
LIN {X 247.534,Y 151.085,Z 94.636,A -148.602,B 90.000,C 0.000} C_DIS
LIN {X 247.527,Y 151.098,Z 94.750,A -148.599,B 90.000,C 0.000} C_DIS
LIN {X 247.457,Y 151.211,Z 95.376,A -148.573,B 90.000,C 0.000} C_DIS
LIN {X 247.379,Y 151.340,Z 95.891,A -148.543,B 90.000,C 0.000} C_DIS
LIN {X 247.359,Y 151.372,Z 96.002,A -148.535,B 90.000,C 0.000} C_DIS
LIN {X 247.343,Y 151.398,Z 96.060,A -148.529,B 90.000,C 0.000} C_DIS
LIN {X 247.168,Y 151.683,Z 98.263,A -148.463,B 90.000,C 0.000} C_DIS
LIN {X 247.141,Y 151.727,Z 98.448,A -148.453,B 90.000,C 0.000} C_DIS
LIN {X 247.033,Y 151.903,Z 100.940,A -148.412,B 90.000,C 0.000} C_DIS
LIN {X 247.036,Y 151.899,Z 103.440,A -148.413,B 90.000,C 0.000} C_DIS
LIN {X 247.066,Y 151.850,Z 105.939,A -148.424,B 90.000,C 0.000} C_DIS
LIN {X 247.209,Y 151.617,Z 108.424,A -148.479,B 90.000,C 0.000} C_DIS
LIN {X 247.436,Y 151.246,Z 110.885,A -148.565,B 90.000,C 0.000} C_DIS
LIN {X 247.723,Y 150.776,Z 113.324,A -148.673,B 90.000,C 0.000} C_DIS
LIN {X 248.114,Y 150.131,Z 115.707,A -148.822,B 90.000,C 0.000} C_DIS
LIN {X 248.578,Y 149.361,Z 118.040,A -149.000,B 90.000,C 0.000} C_DIS
LIN {X 249.141,Y 148.421,Z 120.287,A -149.216,B 90.000,C 0.000} C_DIS
LIN {X 249.468,Y 147.871,Z 121.410,A -149.343,B 90.000,C 0.000} C_DIS
LIN {X 249.616,Y 147.621,Z 121.795,A -149.400,B 90.000,C 0.000} C_DIS
LIN {X 249.732,Y 147.425,Z 122.205,A -149.445,B 90.000,C 0.000} C_DIS
LIN {X 249.818,Y 147.278,Z 122.400,A -149.479,B 90.000,C 0.000} C_DIS
LIN {X 249.869,Y 147.192,Z 122.563,A -149.499,B 90.000,C 0.000} C_DIS
LIN {X 250.056,Y 146.873,Z 123.020,A -149.572,B 90.000,C 0.000} C_DIS
LIN {X 250.107,Y 146.787,Z 123.176,A -149.591,B 90.000,C 0.000} C_DIS
LIN {X 250.193,Y 146.640,Z 123.395,A -149.625,B 90.000,C 0.000} C_DIS
LIN {X 250.236,Y 146.567,Z 123.483,A -149.642,B 90.000,C 0.000} C_DIS
LIN {X 250.281,Y 146.491,Z 123.554,A -149.659,B 90.000,C 0.000} C_DIS
LIN {X 250.468,Y 146.171,Z 124.039,A -149.732,B 90.000,C 0.000} C_DIS
LIN {X 251.279,Y 144.771,Z 125.374,A -150.052,B 90.000,C 0.000} C_DIS
LIN {X 251.308,Y 144.722,Z 125.389,A -150.063,B 90.000,C 0.000} C_DIS
LIN {X 251.336,Y 144.672,Z 125.414,A -150.075,B 90.000,C 0.000} C_DIS
LIN {X 251.421,Y 144.524,Z 125.534,A -150.108,B 90.000,C 0.000} C_DIS
LIN {X 251.478,Y 144.426,Z 125.583,A -150.131,B 90.000,C 0.000} C_DIS
LIN {X 251.846,Y 143.784,Z 125.998,A -150.277,B 90.000,C 0.000} C_DIS
LIN {X 251.902,Y 143.685,Z 126.027,A -150.300,B 90.000,C 0.000} C_DIS
LIN {X 252.486,Y 142.656,Z 126.398,A -150.533,B 90.000,C 0.000} C_DIS
LIN {X 253.660,Y 140.557,Z 125.714,A -151.008,B 90.000,C 0.000} C_DIS
LIN {X 254.803,Y 138.475,Z 124.935,A -151.478,B 90.000,C 0.000} C_DIS
LIN {X 255.920,Y 136.400,Z 124.100,A -151.943,B 90.000,C 0.000} C_DIS
LIN {X 257.009,Y 134.338,Z 123.200,A -152.404,B 90.000,C 0.000} C_DIS
LIN {X 258.062,Y 132.303,Z 122.199,A -152.857,B 90.000,C 0.000} C_DIS
LIN {X 258.519,Y 131.407,Z 121.667,A -153.055,B 90.000,C 0.000} C_DIS
RET=EKI_SetBool("oxy","torchState",FALSE)
RET = EKI_Send("oxy","torchState")
PTP {X 256.736,Y 130.501,Z 121.667,A -153.055,B 90.000,C 0.000}
PTP {X 240.690,Y 122.345,Z 121.667,A -153.055,B 90.000,C 0.000}
PTP {X 236.352,Y 130.529,Z 136.457,A -151.090,B 90.000,C 0.000}
PTP {X 252.108,Y 139.231,Z 136.457,A -151.090,B 90.000,C 0.000}
WAIT SEC 2
RET=EKI_SetBool("oxy","torchState",TRUE)
RET = EKI_Send("oxy","torchState")
LIN {X 253.859,Y 140.198,Z 136.457,A -151.090,B 90.000,C 0.000} C_DIS
LIN {X 254.703,Y 138.660,Z 137.764,A -151.436,B 90.000,C 0.000} C_DIS
LIN {X 255.496,Y 137.193,Z 138.973,A -151.766,B 90.000,C 0.000} C_DIS
LIN {X 255.537,Y 137.116,Z 139.072,A -151.783,B 90.000,C 0.000} C_DIS
LIN {X 255.849,Y 136.534,Z 139.584,A -151.913,B 90.000,C 0.000} C_DIS
LIN {X 255.901,Y 136.435,Z 139.655,A -151.936,B 90.000,C 0.000} C_DIS
LIN {X 256.183,Y 135.905,Z 140.162,A -152.054,B 90.000,C 0.000} C_DIS
LIN {X 256.272,Y 135.737,Z 140.280,A -152.092,B 90.000,C 0.000} C_DIS
LIN {X 256.313,Y 135.660,Z 140.381,A -152.109,B 90.000,C 0.000} C_DIS
LIN {X 257.199,Y 133.973,Z 142.000,A -152.485,B 90.000,C 0.000} C_DIS
LIN {X 257.250,Y 133.874,Z 142.088,A -152.507,B 90.000,C 0.000} C_DIS
LIN {X 258.058,Y 132.309,Z 143.861,A -152.855,B 90.000,C 0.000} C_DIS
LIN {X 258.101,Y 132.226,Z 143.955,A -152.874,B 90.000,C 0.000} C_DIS
LIN {X 258.315,Y 131.808,Z 144.527,A -152.966,B 90.000,C 0.000} C_DIS
LIN {X 258.360,Y 131.720,Z 144.693,A -152.986,B 90.000,C 0.000} C_DIS
LIN {X 258.383,Y 131.675,Z 144.737,A -152.996,B 90.000,C 0.000} C_DIS
LIN {X 258.725,Y 131.001,Z 145.980,A -153.145,B 90.000,C 0.000} C_DIS
LIN {X 258.747,Y 130.957,Z 148.176,A -153.155,B 90.000,C 0.000} C_DIS
LIN {X 258.657,Y 131.135,Z 149.829,A -153.116,B 90.000,C 0.000} C_DIS
LIN {X 258.642,Y 131.165,Z 149.882,A -153.109,B 90.000,C 0.000} C_DIS
LIN {X 258.600,Y 131.249,Z 150.224,A -153.091,B 90.000,C 0.000} C_DIS
LIN {X 258.570,Y 131.307,Z 150.622,A -153.078,B 90.000,C 0.000} C_DIS
LIN {X 258.436,Y 131.572,Z 151.305,A -153.019,B 90.000,C 0.000} C_DIS
LIN {X 258.422,Y 131.598,Z 151.524,A -153.013,B 90.000,C 0.000} C_DIS
LIN {X 258.153,Y 132.125,Z 152.589,A -152.896,B 90.000,C 0.000} C_DIS
LIN {X 258.129,Y 132.172,Z 152.670,A -152.886,B 90.000,C 0.000} C_DIS
LIN {X 257.913,Y 132.593,Z 153.321,A -152.792,B 90.000,C 0.000} C_DIS
LIN {X 257.830,Y 132.754,Z 153.474,A -152.757,B 90.000,C 0.000} C_DIS
LIN {X 257.765,Y 132.881,Z 153.695,A -152.728,B 90.000,C 0.000} C_DIS
LIN {X 257.434,Y 133.521,Z 154.287,A -152.586,B 90.000,C 0.000} C_DIS
LIN {X 257.161,Y 134.046,Z 154.713,A -152.469,B 90.000,C 0.000} C_DIS
LIN {X 256.739,Y 134.853,Z 155.175,A -152.289,B 90.000,C 0.000} C_DIS
LIN {X 255.608,Y 136.984,Z 155.830,A -151.813,B 90.000,C 0.000} C_DIS
LIN {X 255.544,Y 137.104,Z 155.859,A -151.786,B 90.000,C 0.000} C_DIS
LIN {X 254.829,Y 138.428,Z 156.000,A -151.488,B 90.000,C 0.000} C_DIS
LIN {X 254.658,Y 138.742,Z 155.985,A -151.418,B 90.000,C 0.000} C_DIS
LIN {X 254.767,Y 138.542,Z 155.230,A -151.463,B 90.000,C 0.000} C_DIS
LIN {X 254.791,Y 138.497,Z 154.548,A -151.473,B 90.000,C 0.000} C_DIS
LIN {X 254.751,Y 138.570,Z 153.707,A -151.456,B 90.000,C 0.000} C_DIS
LIN {X 254.536,Y 138.965,Z 152.811,A -151.367,B 90.000,C 0.000} C_DIS
LIN {X 254.328,Y 139.345,Z 152.299,A -151.282,B 90.000,C 0.000} C_DIS
LIN {X 254.038,Y 139.874,Z 151.814,A -151.163,B 90.000,C 0.000} C_DIS
LIN {X 253.934,Y 140.063,Z 151.701,A -151.120,B 90.000,C 0.000} C_DIS
LIN {X 253.297,Y 141.211,Z 151.390,A -150.861,B 90.000,C 0.000} C_DIS
LIN {X 252.860,Y 141.993,Z 151.519,A -150.684,B 90.000,C 0.000} C_DIS
LIN {X 252.505,Y 142.622,Z 151.781,A -150.541,B 90.000,C 0.000} C_DIS
LIN {X 252.419,Y 142.775,Z 151.874,A -150.506,B 90.000,C 0.000} C_DIS
LIN {X 252.362,Y 142.876,Z 151.959,A -150.483,B 90.000,C 0.000} C_DIS
LIN {X 251.986,Y 143.537,Z 152.711,A -150.333,B 90.000,C 0.000} C_DIS
LIN {X 251.836,Y 143.801,Z 153.202,A -150.273,B 90.000,C 0.000} C_DIS
LIN {X 251.734,Y 143.979,Z 153.820,A -150.233,B 90.000,C 0.000} C_DIS
LIN {X 251.693,Y 144.051,Z 154.476,A -150.216,B 90.000,C 0.000} C_DIS
LIN {X 251.746,Y 143.958,Z 155.460,A -150.237,B 90.000,C 0.000} C_DIS
LIN {X 251.756,Y 143.940,Z 155.515,A -150.241,B 90.000,C 0.000} C_DIS
LIN {X 251.800,Y 143.864,Z 155.652,A -150.259,B 90.000,C 0.000} C_DIS
LIN {X 251.833,Y 143.806,Z 155.872,A -150.272,B 90.000,C 0.000} C_DIS
LIN {X 251.791,Y 143.880,Z 155.986,A -150.255,B 90.000,C 0.000} C_DIS
LIN {X 251.078,Y 145.119,Z 155.774,A -149.973,B 90.000,C 0.000} C_DIS
LIN {X 251.052,Y 145.165,Z 155.739,A -149.962,B 90.000,C 0.000} C_DIS
LIN {X 250.995,Y 145.264,Z 155.702,A -149.940,B 90.000,C 0.000} C_DIS
LIN {X 250.852,Y 145.510,Z 155.669,A -149.884,B 90.000,C 0.000} C_DIS
LIN {X 250.681,Y 145.805,Z 155.575,A -149.816,B 90.000,C 0.000} C_DIS
LIN {X 250.652,Y 145.855,Z 155.544,A -149.805,B 90.000,C 0.000} C_DIS
LIN {X 250.298,Y 146.461,Z 155.394,A -149.666,B 90.000,C 0.000} C_DIS
LIN {X 250.240,Y 146.560,Z 155.354,A -149.644,B 90.000,C 0.000} C_DIS
LIN {X 250.107,Y 146.788,Z 155.295,A -149.591,B 90.000,C 0.000} C_DIS
LIN {X 249.297,Y 148.159,Z 154.654,A -149.277,B 90.000,C 0.000} C_DIS
LIN {X 249.275,Y 148.196,Z 154.614,A -149.268,B 90.000,C 0.000} C_DIS
LIN {X 249.062,Y 148.554,Z 154.491,A -149.186,B 90.000,C 0.000} C_DIS
LIN {X 249.035,Y 148.599,Z 154.425,A -149.175,B 90.000,C 0.000} C_DIS
LIN {X 249.018,Y 148.628,Z 154.392,A -149.169,B 90.000,C 0.000} C_DIS
LIN {X 248.633,Y 149.271,Z 154.036,A -149.021,B 90.000,C 0.000} C_DIS
LIN {X 248.532,Y 149.439,Z 153.890,A -148.982,B 90.000,C 0.000} C_DIS
LIN {X 248.345,Y 149.749,Z 153.695,A -148.910,B 90.000,C 0.000} C_DIS
LIN {X 248.286,Y 149.847,Z 153.595,A -148.888,B 90.000,C 0.000} C_DIS
LIN {X 248.146,Y 150.078,Z 153.467,A -148.835,B 90.000,C 0.000} C_DIS
LIN {X 247.656,Y 150.886,Z 152.727,A -148.648,B 90.000,C 0.000} C_DIS
LIN {X 247.624,Y 150.938,Z 152.667,A -148.636,B 90.000,C 0.000} C_DIS
LIN {X 247.597,Y 150.983,Z 152.639,A -148.625,B 90.000,C 0.000} C_DIS
LIN {X 247.461,Y 151.206,Z 152.382,A -148.574,B 90.000,C 0.000} C_DIS
LIN {X 247.426,Y 151.263,Z 152.293,A -148.561,B 90.000,C 0.000} C_DIS
LIN {X 247.209,Y 151.617,Z 151.914,A -148.478,B 90.000,C 0.000} C_DIS
LIN {X 246.724,Y 152.405,Z 150.862,A -148.296,B 90.000,C 0.000} C_DIS
LIN {X 246.672,Y 152.490,Z 150.693,A -148.276,B 90.000,C 0.000} C_DIS
LIN {X 246.403,Y 152.924,Z 149.882,A -148.175,B 90.000,C 0.000} C_DIS
LIN {X 246.312,Y 153.070,Z 149.482,A -148.141,B 90.000,C 0.000} C_DIS
LIN {X 246.372,Y 152.973,Z 149.411,A -148.164,B 90.000,C 0.000} C_DIS
LIN {X 246.612,Y 152.586,Z 149.525,A -148.254,B 90.000,C 0.000} C_DIS
LIN {X 246.856,Y 152.192,Z 149.564,A -148.345,B 90.000,C 0.000} C_DIS
LIN {X 247.179,Y 151.666,Z 149.465,A -148.467,B 90.000,C 0.000} C_DIS
LIN {X 247.342,Y 151.400,Z 149.311,A -148.529,B 90.000,C 0.000} C_DIS
LIN {X 247.452,Y 151.220,Z 149.114,A -148.570,B 90.000,C 0.000} C_DIS
LIN {X 247.507,Y 151.131,Z 148.972,A -148.591,B 90.000,C 0.000} C_DIS
LIN {X 247.580,Y 151.010,Z 148.594,A -148.619,B 90.000,C 0.000} C_DIS
LIN {X 247.611,Y 150.960,Z 147.948,A -148.631,B 90.000,C 0.000} C_DIS
LIN {X 247.579,Y 151.011,Z 147.497,A -148.619,B 90.000,C 0.000} C_DIS
LIN {X 247.497,Y 151.147,Z 147.345,A -148.587,B 90.000,C 0.000} C_DIS
LIN {X 246.612,Y 152.586,Z 145.892,A -148.254,B 90.000,C 0.000} C_DIS
LIN {X 246.584,Y 152.631,Z 145.869,A -148.243,B 90.000,C 0.000} C_DIS
LIN {X 246.536,Y 152.708,Z 145.783,A -148.225,B 90.000,C 0.000} C_DIS
LIN {X 246.502,Y 152.764,Z 145.692,A -148.212,B 90.000,C 0.000} C_DIS
LIN {X 246.281,Y 153.120,Z 145.317,A -148.130,B 90.000,C 0.000} C_DIS
LIN {X 245.731,Y 154.001,Z 144.061,A -147.924,B 90.000,C 0.000} C_DIS
LIN {X 245.680,Y 154.082,Z 143.965,A -147.906,B 90.000,C 0.000} C_DIS
LIN {X 245.490,Y 154.385,Z 143.446,A -147.835,B 90.000,C 0.000} C_DIS
LIN {X 244.884,Y 155.345,Z 141.219,A -147.611,B 90.000,C 0.000} C_DIS
LIN {X 244.661,Y 155.695,Z 140.048,A -147.528,B 90.000,C 0.000} C_DIS
LIN {X 244.568,Y 155.841,Z 139.247,A -147.494,B 90.000,C 0.000} C_DIS
LIN {X 244.492,Y 155.961,Z 137.947,A -147.466,B 90.000,C 0.000} C_DIS
LIN {X 244.503,Y 155.943,Z 136.842,A -147.471,B 90.000,C 0.000} C_DIS
LIN {X 244.582,Y 155.819,Z 136.138,A -147.500,B 90.000,C 0.000} C_DIS
LIN {X 244.629,Y 155.746,Z 136.015,A -147.517,B 90.000,C 0.000} C_DIS
LIN {X 244.707,Y 155.623,Z 136.227,A -147.545,B 90.000,C 0.000} C_DIS
LIN {X 244.834,Y 155.423,Z 136.740,A -147.592,B 90.000,C 0.000} C_DIS
LIN {X 244.997,Y 155.166,Z 137.139,A -147.652,B 90.000,C 0.000} C_DIS
LIN {X 245.710,Y 154.035,Z 138.273,A -147.916,B 90.000,C 0.000} C_DIS
LIN {X 246.367,Y 152.982,Z 139.015,A -148.162,B 90.000,C 0.000} C_DIS
LIN {X 246.402,Y 152.925,Z 139.071,A -148.175,B 90.000,C 0.000} C_DIS
LIN {X 246.552,Y 152.683,Z 139.249,A -148.231,B 90.000,C 0.000} C_DIS
LIN {X 246.574,Y 152.647,Z 139.291,A -148.240,B 90.000,C 0.000} C_DIS
LIN {X 246.793,Y 152.293,Z 139.414,A -148.322,B 90.000,C 0.000} C_DIS
LIN {X 246.821,Y 152.247,Z 139.474,A -148.332,B 90.000,C 0.000} C_DIS
LIN {X 246.881,Y 152.151,Z 139.518,A -148.355,B 90.000,C 0.000} C_DIS
LIN {X 246.960,Y 152.022,Z 139.608,A -148.385,B 90.000,C 0.000} C_DIS
LIN {X 247.093,Y 151.807,Z 139.611,A -148.435,B 90.000,C 0.000} C_DIS
LIN {X 247.158,Y 151.700,Z 139.471,A -148.459,B 90.000,C 0.000} C_DIS
LIN {X 247.272,Y 151.515,Z 139.364,A -148.502,B 90.000,C 0.000} C_DIS
LIN {X 247.957,Y 150.390,Z 138.914,A -148.763,B 90.000,C 0.000} C_DIS
LIN {X 249.227,Y 148.277,Z 138.498,A -149.250,B 90.000,C 0.000} C_DIS
LIN {X 250.490,Y 146.124,Z 138.354,A -149.743,B 90.000,C 0.000} C_DIS
LIN {X 251.736,Y 143.957,Z 138.340,A -150.237,B 90.000,C 0.000} C_DIS
LIN {X 252.975,Y 141.786,Z 138.365,A -150.730,B 90.000,C 0.000} C_DIS
LIN {X 253.410,Y 141.008,Z 138.421,A -150.907,B 90.000,C 0.000} C_DIS
LIN {X 253.521,Y 140.809,Z 138.375,A -150.951,B 90.000,C 0.000} C_DIS
LIN {X 253.496,Y 140.854,Z 138.357,A -150.941,B 90.000,C 0.000} C_DIS
LIN {X 253.410,Y 141.008,Z 138.247,A -150.907,B 90.000,C 0.000} C_DIS
LIN {X 253.382,Y 141.058,Z 138.226,A -150.895,B 90.000,C 0.000} C_DIS
LIN {X 252.663,Y 142.342,Z 137.024,A -150.605,B 90.000,C 0.000} C_DIS
LIN {X 252.577,Y 142.495,Z 136.811,A -150.570,B 90.000,C 0.000} C_DIS
LIN {X 252.492,Y 142.646,Z 136.660,A -150.536,B 90.000,C 0.000} C_DIS
LIN {X 252.408,Y 142.795,Z 136.428,A -150.502,B 90.000,C 0.000} C_DIS
LIN {X 252.324,Y 142.943,Z 136.267,A -150.468,B 90.000,C 0.000} C_DIS
LIN {X 252.176,Y 143.203,Z 135.822,A -150.409,B 90.000,C 0.000} C_DIS
LIN {X 252.127,Y 143.290,Z 135.628,A -150.389,B 90.000,C 0.000} C_DIS
LIN {X 252.043,Y 143.438,Z 135.404,A -150.356,B 90.000,C 0.000} C_DIS
LIN {X 251.529,Y 144.338,Z 133.129,A -150.151,B 90.000,C 0.000} C_DIS
LIN {X 251.374,Y 144.606,Z 131.991,A -150.090,B 90.000,C 0.000} C_DIS
LIN {X 251.363,Y 144.626,Z 131.479,A -150.085,B 90.000,C 0.000} C_DIS
LIN {X 251.677,Y 144.078,Z 132.984,A -150.210,B 90.000,C 0.000} C_DIS
LIN {X 252.611,Y 142.435,Z 134.621,A -150.583,B 90.000,C 0.000} C_DIS
LIN {X 252.754,Y 142.180,Z 134.821,A -150.641,B 90.000,C 0.000} C_DIS
LIN {X 252.813,Y 142.076,Z 134.919,A -150.665,B 90.000,C 0.000} C_DIS
LIN {X 252.855,Y 142.002,Z 134.963,A -150.682,B 90.000,C 0.000} C_DIS
LIN {X 253.462,Y 140.916,Z 135.886,A -150.927,B 90.000,C 0.000} C_DIS
LIN {X 253.509,Y 140.830,Z 135.986,A -150.947,B 90.000,C 0.000} C_DIS
LIN {X 253.704,Y 140.479,Z 136.274,A -151.026,B 90.000,C 0.000} C_DIS
LIN {X 253.859,Y 140.198,Z 136.457,A -151.090,B 90.000,C 0.000} C_DIS
RET=EKI_SetBool("oxy","torchState",FALSE)
RET = EKI_Send("oxy","torchState")
PTP {X 252.108,Y 139.231,Z 136.457,A -151.090,B 90.000,C 0.000}
PTP {X 236.352,Y 130.529,Z 136.457,A -151.090,B 90.000,C 0.000}
PTP {X 235.573,Y 131.929,Z 159.730,A -150.750,B 90.000,C 0.000}
PTP {X 251.278,Y 140.724,Z 159.730,A -150.750,B 90.000,C 0.000}
WAIT SEC 2
RET=EKI_SetBool("oxy","torchState",TRUE)
RET = EKI_Send("oxy","torchState")
LIN {X 253.023,Y 141.701,Z 159.730,A -150.750,B 90.000,C 0.000} C_DIS
LIN {X 252.981,Y 141.776,Z 159.717,A -150.733,B 90.000,C 0.000} C_DIS
LIN {X 251.870,Y 143.741,Z 160.791,A -150.287,B 90.000,C 0.000} C_DIS
LIN {X 250.710,Y 145.755,Z 161.712,A -149.828,B 90.000,C 0.000} C_DIS
LIN {X 249.932,Y 147.084,Z 162.233,A -149.523,B 90.000,C 0.000} C_DIS
LIN {X 249.818,Y 147.278,Z 162.273,A -149.479,B 90.000,C 0.000} C_DIS
LIN {X 249.630,Y 147.598,Z 162.421,A -149.406,B 90.000,C 0.000} C_DIS
LIN {X 249.411,Y 147.967,Z 162.483,A -149.321,B 90.000,C 0.000} C_DIS
LIN {X 249.355,Y 148.061,Z 162.543,A -149.299,B 90.000,C 0.000} C_DIS
LIN {X 248.091,Y 150.169,Z 163.000,A -148.814,B 90.000,C 0.000} C_DIS
LIN {X 246.972,Y 152.003,Z 163.223,A -148.389,B 90.000,C 0.000} C_DIS
LIN {X 246.936,Y 152.062,Z 163.199,A -148.375,B 90.000,C 0.000} C_DIS
LIN {X 246.702,Y 152.441,Z 163.187,A -148.287,B 90.000,C 0.000} C_DIS
LIN {X 246.677,Y 152.482,Z 163.162,A -148.278,B 90.000,C 0.000} C_DIS
LIN {X 245.596,Y 154.216,Z 163.126,A -147.874,B 90.000,C 0.000} C_DIS
LIN {X 245.141,Y 154.938,Z 163.003,A -147.706,B 90.000,C 0.000} C_DIS
LIN {X 243.834,Y 156.986,Z 162.415,A -147.226,B 90.000,C 0.000} C_DIS
LIN {X 243.045,Y 158.207,Z 161.930,A -146.938,B 90.000,C 0.000} C_DIS
LIN {X 242.982,Y 158.302,Z 161.898,A -146.916,B 90.000,C 0.000} C_DIS
LIN {X 242.687,Y 158.755,Z 161.659,A -146.809,B 90.000,C 0.000} C_DIS
LIN {X 242.638,Y 158.829,Z 161.634,A -146.791,B 90.000,C 0.000} C_DIS
LIN {X 242.609,Y 158.874,Z 161.606,A -146.781,B 90.000,C 0.000} C_DIS
LIN {X 242.565,Y 158.942,Z 161.546,A -146.765,B 90.000,C 0.000} C_DIS
LIN {X 242.172,Y 159.539,Z 161.203,A -146.624,B 90.000,C 0.000} C_DIS
LIN {X 242.133,Y 159.599,Z 161.147,A -146.610,B 90.000,C 0.000} C_DIS
LIN {X 241.426,Y 160.666,Z 160.466,A -146.357,B 90.000,C 0.000} C_DIS
LIN {X 241.331,Y 160.808,Z 160.327,A -146.323,B 90.000,C 0.000} C_DIS
LIN {X 240.533,Y 162.000,Z 159.327,A -146.040,B 90.000,C 0.000} C_DIS
LIN {X 240.500,Y 162.049,Z 159.242,A -146.028,B 90.000,C 0.000} C_DIS
LIN {X 240.452,Y 162.120,Z 159.157,A -146.011,B 90.000,C 0.000} C_DIS
LIN {X 240.385,Y 162.219,Z 159.058,A -145.987,B 90.000,C 0.000} C_DIS
LIN {X 240.081,Y 162.668,Z 158.670,A -145.880,B 90.000,C 0.000} C_DIS
LIN {X 239.990,Y 162.802,Z 158.502,A -145.848,B 90.000,C 0.000} C_DIS
LIN {X 239.926,Y 162.897,Z 158.413,A -145.826,B 90.000,C 0.000} C_DIS
LIN {X 239.878,Y 162.968,Z 158.360,A -145.809,B 90.000,C 0.000} C_DIS
LIN {X 239.830,Y 163.038,Z 158.275,A -145.792,B 90.000,C 0.000} C_DIS
LIN {X 239.799,Y 163.084,Z 158.189,A -145.781,B 90.000,C 0.000} C_DIS
LIN {X 239.317,Y 163.790,Z 157.450,A -145.612,B 90.000,C 0.000} C_DIS
LIN {X 239.183,Y 163.986,Z 157.165,A -145.565,B 90.000,C 0.000} C_DIS
LIN {X 238.592,Y 164.845,Z 156.048,A -145.359,B 90.000,C 0.000} C_DIS
LIN {X 238.543,Y 164.915,Z 155.936,A -145.342,B 90.000,C 0.000} C_DIS
LIN {X 238.446,Y 165.056,Z 155.777,A -145.308,B 90.000,C 0.000} C_DIS
LIN {X 238.349,Y 165.196,Z 155.545,A -145.275,B 90.000,C 0.000} C_DIS
LIN {X 238.252,Y 165.336,Z 155.379,A -145.241,B 90.000,C 0.000} C_DIS
LIN {X 238.154,Y 165.477,Z 155.176,A -145.207,B 90.000,C 0.000} C_DIS
LIN {X 238.097,Y 165.558,Z 155.007,A -145.188,B 90.000,C 0.000} C_DIS
LIN {X 237.797,Y 165.990,Z 154.383,A -145.084,B 90.000,C 0.000} C_DIS
LIN {X 237.732,Y 166.084,Z 154.169,A -145.061,B 90.000,C 0.000} C_DIS
LIN {X 237.634,Y 166.223,Z 154.016,A -145.027,B 90.000,C 0.000} C_DIS
LIN {X 237.503,Y 166.410,Z 153.626,A -144.982,B 90.000,C 0.000} C_DIS
LIN {X 237.473,Y 166.453,Z 153.606,A -144.972,B 90.000,C 0.000} C_DIS
LIN {X 237.372,Y 166.597,Z 153.325,A -144.937,B 90.000,C 0.000} C_DIS
LIN {X 237.251,Y 166.770,Z 153.091,A -144.896,B 90.000,C 0.000} C_DIS
LIN {X 237.239,Y 166.786,Z 152.991,A -144.892,B 90.000,C 0.000} C_DIS
LIN {X 236.881,Y 167.294,Z 152.139,A -144.769,B 90.000,C 0.000} C_DIS
LIN {X 236.153,Y 168.320,Z 149.978,A -144.520,B 90.000,C 0.000} C_DIS
LIN {X 235.922,Y 168.644,Z 149.314,A -144.442,B 90.000,C 0.000} C_DIS
LIN {X 235.255,Y 169.573,Z 147.091,A -144.216,B 90.000,C 0.000} C_DIS
LIN {X 234.651,Y 170.408,Z 144.813,A -144.012,B 90.000,C 0.000} C_DIS
LIN {X 234.088,Y 171.180,Z 142.503,A -143.823,B 90.000,C 0.000} C_DIS
LIN {X 233.573,Y 171.882,Z 140.159,A -143.651,B 90.000,C 0.000} C_DIS
LIN {X 233.064,Y 172.572,Z 137.811,A -143.482,B 90.000,C 0.000} C_DIS
LIN {X 232.915,Y 172.774,Z 137.268,A -143.432,B 90.000,C 0.000} C_DIS
LIN {X 232.915,Y 172.774,Z 137.268,A -143.432,B 90.000,C 0.000} C_DIS
LIN {X 232.835,Y 172.881,Z 137.148,A -143.406,B 90.000,C 0.000} C_DIS
LIN {X 232.733,Y 173.018,Z 137.522,A -143.372,B 90.000,C 0.000} C_DIS
LIN {X 232.729,Y 173.024,Z 137.594,A -143.371,B 90.000,C 0.000} C_DIS
LIN {X 232.593,Y 173.207,Z 138.289,A -143.326,B 90.000,C 0.000} C_DIS
LIN {X 232.522,Y 173.302,Z 138.961,A -143.302,B 90.000,C 0.000} C_DIS
LIN {X 232.502,Y 173.328,Z 139.015,A -143.296,B 90.000,C 0.000} C_DIS
LIN {X 232.484,Y 173.353,Z 139.158,A -143.290,B 90.000,C 0.000} C_DIS
LIN {X 232.479,Y 173.359,Z 139.300,A -143.288,B 90.000,C 0.000} C_DIS
LIN {X 232.449,Y 173.399,Z 139.485,A -143.278,B 90.000,C 0.000} C_DIS
LIN {X 232.319,Y 173.575,Z 141.838,A -143.235,B 90.000,C 0.000} C_DIS
LIN {X 232.260,Y 173.652,Z 141.974,A -143.216,B 90.000,C 0.000} C_DIS
LIN {X 232.208,Y 173.723,Z 141.861,A -143.198,B 90.000,C 0.000} C_DIS
LIN {X 232.160,Y 173.787,Z 141.779,A -143.183,B 90.000,C 0.000} C_DIS
LIN {X 232.129,Y 173.827,Z 141.786,A -143.173,B 90.000,C 0.000} C_DIS
LIN {X 231.695,Y 174.405,Z 139.392,A -143.030,B 90.000,C 0.000} C_DIS
LIN {X 231.377,Y 174.828,Z 137.496,A -142.925,B 90.000,C 0.000} C_DIS
LIN {X 231.343,Y 174.873,Z 137.422,A -142.914,B 90.000,C 0.000} C_DIS
LIN {X 231.306,Y 174.921,Z 137.607,A -142.902,B 90.000,C 0.000} C_DIS
LIN {X 231.228,Y 175.024,Z 140.104,A -142.877,B 90.000,C 0.000} C_DIS
LIN {X 231.167,Y 175.105,Z 142.602,A -142.857,B 90.000,C 0.000} C_DIS
LIN {X 231.131,Y 175.153,Z 145.101,A -142.845,B 90.000,C 0.000} C_DIS
LIN {X 231.086,Y 175.213,Z 147.600,A -142.830,B 90.000,C 0.000} C_DIS
LIN {X 231.062,Y 175.244,Z 148.631,A -142.822,B 90.000,C 0.000} C_DIS
LIN {X 231.067,Y 175.236,Z 149.256,A -142.824,B 90.000,C 0.000} C_DIS
LIN {X 231.084,Y 175.215,Z 151.644,A -142.830,B 90.000,C 0.000} C_DIS
LIN {X 231.074,Y 175.227,Z 151.703,A -142.826,B 90.000,C 0.000} C_DIS
LIN {X 231.084,Y 175.215,Z 152.881,A -142.829,B 90.000,C 0.000} C_DIS
LIN {X 231.066,Y 175.238,Z 153.012,A -142.824,B 90.000,C 0.000} C_DIS
LIN {X 231.052,Y 175.257,Z 153.072,A -142.819,B 90.000,C 0.000} C_DIS
LIN {X 231.117,Y 175.171,Z 155.395,A -142.840,B 90.000,C 0.000} C_DIS
LIN {X 231.088,Y 175.210,Z 155.522,A -142.831,B 90.000,C 0.000} C_DIS
LIN {X 231.166,Y 175.107,Z 158.019,A -142.856,B 90.000,C 0.000} C_DIS
LIN {X 231.229,Y 175.023,Z 160.517,A -142.877,B 90.000,C 0.000} C_DIS
LIN {X 231.272,Y 174.966,Z 161.532,A -142.891,B 90.000,C 0.000} C_DIS
LIN {X 231.275,Y 174.962,Z 161.959,A -142.892,B 90.000,C 0.000} C_DIS
LIN {X 231.394,Y 174.805,Z 164.106,A -142.931,B 90.000,C 0.000} C_DIS
LIN {X 231.385,Y 174.817,Z 164.163,A -142.928,B 90.000,C 0.000} C_DIS
LIN {X 231.445,Y 174.738,Z 165.643,A -142.948,B 90.000,C 0.000} C_DIS
LIN {X 231.604,Y 174.527,Z 168.129,A -143.000,B 90.000,C 0.000} C_DIS
LIN {X 231.776,Y 174.299,Z 170.612,A -143.056,B 90.000,C 0.000} C_DIS
LIN {X 231.976,Y 174.032,Z 173.090,A -143.122,B 90.000,C 0.000} C_DIS
LIN {X 232.205,Y 173.727,Z 175.560,A -143.197,B 90.000,C 0.000} C_DIS
LIN {X 232.422,Y 173.436,Z 177.684,A -143.269,B 90.000,C 0.000} C_DIS
LIN {X 232.451,Y 173.396,Z 177.822,A -143.279,B 90.000,C 0.000} C_DIS
LIN {X 232.508,Y 173.321,Z 178.416,A -143.298,B 90.000,C 0.000} C_DIS
LIN {X 232.639,Y 173.145,Z 179.021,A -143.341,B 90.000,C 0.000} C_DIS
LIN {X 232.843,Y 172.870,Z 179.245,A -143.409,B 90.000,C 0.000} C_DIS
LIN {X 232.869,Y 172.836,Z 179.288,A -143.417,B 90.000,C 0.000} C_DIS
LIN {X 233.413,Y 172.100,Z 179.711,A -143.598,B 90.000,C 0.000} C_DIS
LIN {X 233.455,Y 172.042,Z 179.721,A -143.612,B 90.000,C 0.000} C_DIS
LIN {X 233.486,Y 172.001,Z 179.743,A -143.622,B 90.000,C 0.000} C_DIS
LIN {X 233.655,Y 171.771,Z 179.921,A -143.679,B 90.000,C 0.000} C_DIS
LIN {X 233.790,Y 171.588,Z 179.975,A -143.723,B 90.000,C 0.000} C_DIS
LIN {X 234.394,Y 170.761,Z 180.461,A -143.926,B 90.000,C 0.000} C_DIS
LIN {X 234.436,Y 170.704,Z 180.476,A -143.940,B 90.000,C 0.000} C_DIS
LIN {X 235.660,Y 169.009,Z 181.235,A -144.353,B 90.000,C 0.000} C_DIS
LIN {X 236.124,Y 168.361,Z 181.518,A -144.510,B 90.000,C 0.000} C_DIS
LIN {X 236.256,Y 168.176,Z 181.553,A -144.555,B 90.000,C 0.000} C_DIS
LIN {X 236.914,Y 167.248,Z 181.850,A -144.780,B 90.000,C 0.000} C_DIS
LIN {X 236.956,Y 167.189,Z 181.884,A -144.794,B 90.000,C 0.000} C_DIS
LIN {X 238.029,Y 165.657,Z 182.223,A -145.164,B 90.000,C 0.000} C_DIS
LIN {X 238.057,Y 165.617,Z 182.259,A -145.174,B 90.000,C 0.000} C_DIS
LIN {X 238.109,Y 165.543,Z 182.291,A -145.191,B 90.000,C 0.000} C_DIS
LIN {X 238.195,Y 165.418,Z 182.293,A -145.221,B 90.000,C 0.000} C_DIS
LIN {X 238.810,Y 164.529,Z 182.463,A -145.435,B 90.000,C 0.000} C_DIS
LIN {X 240.063,Y 162.695,Z 182.618,A -145.874,B 90.000,C 0.000} C_DIS
LIN {X 241.454,Y 160.620,Z 182.527,A -146.367,B 90.000,C 0.000} C_DIS
LIN {X 242.822,Y 158.548,Z 182.236,A -146.858,B 90.000,C 0.000} C_DIS
LIN {X 243.540,Y 157.443,Z 181.977,A -147.118,B 90.000,C 0.000} C_DIS
LIN {X 244.785,Y 155.501,Z 181.014,A -147.574,B 90.000,C 0.000} C_DIS
LIN {X 245.989,Y 153.588,Z 179.946,A -148.021,B 90.000,C 0.000} C_DIS
LIN {X 247.155,Y 151.705,Z 178.787,A -148.458,B 90.000,C 0.000} C_DIS
LIN {X 247.621,Y 150.943,Z 178.276,A -148.635,B 90.000,C 0.000} C_DIS
LIN {X 246.317,Y 153.061,Z 178.533,A -148.143,B 90.000,C 0.000} C_DIS
LIN {X 246.220,Y 153.218,Z 178.475,A -148.107,B 90.000,C 0.000} C_DIS
LIN {X 245.800,Y 153.891,Z 178.505,A -147.950,B 90.000,C 0.000} C_DIS
LIN {X 245.187,Y 154.866,Z 178.423,A -147.722,B 90.000,C 0.000} C_DIS
LIN {X 243.877,Y 156.919,Z 177.858,A -147.241,B 90.000,C 0.000} C_DIS
LIN {X 243.478,Y 157.539,Z 177.649,A -147.096,B 90.000,C 0.000} C_DIS
LIN {X 242.827,Y 158.540,Z 177.119,A -146.860,B 90.000,C 0.000} C_DIS
LIN {X 242.808,Y 158.569,Z 177.094,A -146.853,B 90.000,C 0.000} C_DIS
LIN {X 242.266,Y 159.397,Z 176.651,A -146.657,B 90.000,C 0.000} C_DIS
LIN {X 242.198,Y 159.499,Z 176.571,A -146.633,B 90.000,C 0.000} C_DIS
LIN {X 242.078,Y 159.682,Z 176.460,A -146.590,B 90.000,C 0.000} C_DIS
LIN {X 242.009,Y 159.787,Z 176.364,A -146.565,B 90.000,C 0.000} C_DIS
LIN {X 241.809,Y 160.089,Z 176.168,A -146.494,B 90.000,C 0.000} C_DIS
LIN {X 241.745,Y 160.185,Z 176.070,A -146.471,B 90.000,C 0.000} C_DIS
LIN {X 240.595,Y 161.908,Z 174.670,A -146.062,B 90.000,C 0.000} C_DIS
LIN {X 239.928,Y 162.895,Z 173.779,A -145.826,B 90.000,C 0.000} C_DIS
LIN {X 239.894,Y 162.944,Z 173.712,A -145.814,B 90.000,C 0.000} C_DIS
LIN {X 239.874,Y 162.974,Z 173.681,A -145.807,B 90.000,C 0.000} C_DIS
LIN {X 239.764,Y 163.135,Z 173.563,A -145.769,B 90.000,C 0.000} C_DIS
LIN {X 238.990,Y 164.267,Z 172.413,A -145.498,B 90.000,C 0.000} C_DIS
LIN {X 238.963,Y 164.307,Z 172.334,A -145.488,B 90.000,C 0.000} C_DIS
LIN {X 238.478,Y 165.009,Z 171.532,A -145.320,B 90.000,C 0.000} C_DIS
LIN {X 238.426,Y 165.084,Z 171.478,A -145.302,B 90.000,C 0.000} C_DIS
LIN {X 238.382,Y 165.149,Z 171.417,A -145.286,B 90.000,C 0.000} C_DIS
LIN {X 238.339,Y 165.211,Z 171.326,A -145.271,B 90.000,C 0.000} C_DIS
LIN {X 238.286,Y 165.287,Z 171.245,A -145.253,B 90.000,C 0.000} C_DIS
LIN {X 238.252,Y 165.336,Z 171.216,A -145.241,B 90.000,C 0.000} C_DIS
LIN {X 237.764,Y 166.037,Z 170.252,A -145.072,B 90.000,C 0.000} C_DIS
LIN {X 237.731,Y 166.084,Z 170.223,A -145.061,B 90.000,C 0.000} C_DIS
LIN {X 237.699,Y 166.130,Z 170.202,A -145.050,B 90.000,C 0.000} C_DIS
LIN {X 237.471,Y 166.456,Z 169.671,A -144.971,B 90.000,C 0.000} C_DIS
LIN {X 237.405,Y 166.550,Z 169.634,A -144.949,B 90.000,C 0.000} C_DIS
LIN {X 237.086,Y 167.003,Z 168.960,A -144.839,B 90.000,C 0.000} C_DIS
LIN {X 236.946,Y 167.203,Z 168.601,A -144.791,B 90.000,C 0.000} C_DIS
LIN {X 236.892,Y 167.279,Z 168.509,A -144.772,B 90.000,C 0.000} C_DIS
LIN {X 236.413,Y 167.956,Z 167.395,A -144.609,B 90.000,C 0.000} C_DIS
LIN {X 236.355,Y 168.037,Z 167.199,A -144.589,B 90.000,C 0.000} C_DIS
LIN {X 236.009,Y 168.522,Z 166.283,A -144.471,B 90.000,C 0.000} C_DIS
LIN {X 235.928,Y 168.636,Z 166.098,A -144.444,B 90.000,C 0.000} C_DIS
LIN {X 235.267,Y 169.557,Z 163.870,A -144.220,B 90.000,C 0.000} C_DIS
LIN {X 234.778,Y 170.233,Z 161.513,A -144.055,B 90.000,C 0.000} C_DIS
LIN {X 234.473,Y 170.654,Z 159.068,A -143.952,B 90.000,C 0.000} C_DIS
LIN {X 234.434,Y 170.707,Z 158.189,A -143.939,B 90.000,C 0.000} C_DIS
LIN {X 234.439,Y 170.699,Z 158.119,A -143.941,B 90.000,C 0.000} C_DIS
LIN {X 234.435,Y 170.706,Z 156.426,A -143.939,B 90.000,C 0.000} C_DIS
LIN {X 234.871,Y 170.104,Z 158.812,A -144.086,B 90.000,C 0.000} C_DIS
LIN {X 234.878,Y 170.094,Z 158.851,A -144.089,B 90.000,C 0.000} C_DIS
LIN {X 235.265,Y 169.559,Z 160.067,A -144.219,B 90.000,C 0.000} C_DIS
LIN {X 235.495,Y 169.240,Z 160.621,A -144.297,B 90.000,C 0.000} C_DIS
LIN {X 236.058,Y 168.454,Z 161.781,A -144.488,B 90.000,C 0.000} C_DIS
LIN {X 236.088,Y 168.411,Z 161.805,A -144.498,B 90.000,C 0.000} C_DIS
LIN {X 236.239,Y 168.199,Z 162.057,A -144.550,B 90.000,C 0.000} C_DIS
LIN {X 236.289,Y 168.129,Z 162.172,A -144.567,B 90.000,C 0.000} C_DIS
LIN {X 237.429,Y 166.515,Z 163.704,A -144.957,B 90.000,C 0.000} C_DIS
LIN {X 237.647,Y 166.205,Z 163.894,A -145.032,B 90.000,C 0.000} C_DIS
LIN {X 237.873,Y 165.881,Z 164.163,A -145.110,B 90.000,C 0.000} C_DIS
LIN {X 238.446,Y 165.056,Z 164.699,A -145.308,B 90.000,C 0.000} C_DIS
LIN {X 238.594,Y 164.842,Z 164.846,A -145.360,B 90.000,C 0.000} C_DIS
LIN {X 238.640,Y 164.775,Z 164.901,A -145.376,B 90.000,C 0.000} C_DIS
LIN {X 238.934,Y 164.348,Z 165.147,A -145.478,B 90.000,C 0.000} C_DIS
LIN {X 238.983,Y 164.278,Z 165.200,A -145.495,B 90.000,C 0.000} C_DIS
LIN {X 239.233,Y 163.913,Z 165.417,A -145.583,B 90.000,C 0.000} C_DIS
LIN {X 239.478,Y 163.556,Z 165.601,A -145.668,B 90.000,C 0.000} C_DIS
LIN {X 239.510,Y 163.509,Z 165.614,A -145.679,B 90.000,C 0.000} C_DIS
LIN {X 239.542,Y 163.462,Z 165.646,A -145.691,B 90.000,C 0.000} C_DIS
LIN {X 239.606,Y 163.368,Z 165.683,A -145.713,B 90.000,C 0.000} C_DIS
LIN {X 239.670,Y 163.274,Z 165.700,A -145.736,B 90.000,C 0.000} C_DIS
LIN {X 239.990,Y 162.803,Z 165.941,A -145.848,B 90.000,C 0.000} C_DIS
LIN {X 240.054,Y 162.709,Z 165.969,A -145.871,B 90.000,C 0.000} C_DIS
LIN {X 240.521,Y 162.018,Z 166.307,A -146.035,B 90.000,C 0.000} C_DIS
LIN {X 240.722,Y 161.718,Z 166.372,A -146.107,B 90.000,C 0.000} C_DIS
LIN {X 241.512,Y 160.536,Z 166.842,A -146.388,B 90.000,C 0.000} C_DIS
LIN {X 241.638,Y 160.346,Z 166.874,A -146.433,B 90.000,C 0.000} C_DIS
LIN {X 241.984,Y 159.824,Z 167.074,A -146.556,B 90.000,C 0.000} C_DIS
LIN {X 242.333,Y 159.294,Z 167.193,A -146.682,B 90.000,C 0.000} C_DIS
LIN {X 242.418,Y 159.165,Z 167.266,A -146.712,B 90.000,C 0.000} C_DIS
LIN {X 242.484,Y 159.064,Z 167.284,A -146.736,B 90.000,C 0.000} C_DIS
LIN {X 242.889,Y 158.445,Z 167.460,A -146.882,B 90.000,C 0.000} C_DIS
LIN {X 242.919,Y 158.400,Z 167.494,A -146.893,B 90.000,C 0.000} C_DIS
LIN {X 243.667,Y 157.247,Z 167.716,A -147.164,B 90.000,C 0.000} C_DIS
LIN {X 243.694,Y 157.204,Z 167.751,A -147.174,B 90.000,C 0.000} C_DIS
LIN {X 243.848,Y 156.965,Z 167.810,A -147.231,B 90.000,C 0.000} C_DIS
LIN {X 243.890,Y 156.900,Z 167.844,A -147.246,B 90.000,C 0.000} C_DIS
LIN {X 244.405,Y 156.096,Z 167.942,A -147.435,B 90.000,C 0.000} C_DIS
LIN {X 244.432,Y 156.055,Z 167.978,A -147.444,B 90.000,C 0.000} C_DIS
LIN {X 244.508,Y 155.935,Z 168.009,A -147.472,B 90.000,C 0.000} C_DIS
LIN {X 244.585,Y 155.815,Z 168.017,A -147.500,B 90.000,C 0.000} C_DIS
LIN {X 244.669,Y 155.683,Z 168.069,A -147.531,B 90.000,C 0.000} C_DIS
LIN {X 245.994,Y 153.579,Z 168.322,A -148.023,B 90.000,C 0.000} C_DIS
LIN {X 247.309,Y 151.453,Z 168.368,A -148.517,B 90.000,C 0.000} C_DIS
LIN {X 248.601,Y 149.323,Z 168.162,A -149.009,B 90.000,C 0.000} C_DIS
LIN {X 249.845,Y 147.232,Z 167.586,A -149.489,B 90.000,C 0.000} C_DIS
LIN {X 250.920,Y 145.393,Z 166.635,A -149.910,B 90.000,C 0.000} C_DIS
LIN {X 250.975,Y 145.298,Z 166.553,A -149.932,B 90.000,C 0.000} C_DIS
LIN {X 251.181,Y 144.941,Z 166.325,A -150.013,B 90.000,C 0.000} C_DIS
LIN {X 251.286,Y 144.759,Z 166.155,A -150.055,B 90.000,C 0.000} C_DIS
LIN {X 251.371,Y 144.613,Z 166.055,A -150.088,B 90.000,C 0.000} C_DIS
LIN {X 252.127,Y 143.290,Z 164.561,A -150.389,B 90.000,C 0.000} C_DIS
LIN {X 252.408,Y 142.795,Z 163.728,A -150.502,B 90.000,C 0.000} C_DIS
LIN {X 252.437,Y 142.742,Z 163.651,A -150.514,B 90.000,C 0.000} C_DIS
LIN {X 252.462,Y 142.699,Z 163.538,A -150.524,B 90.000,C 0.000} C_DIS
LIN {X 252.492,Y 142.646,Z 163.456,A -150.536,B 90.000,C 0.000} C_DIS
LIN {X 252.665,Y 142.340,Z 162.798,A -150.605,B 90.000,C 0.000} C_DIS
LIN {X 252.790,Y 142.117,Z 162.248,A -150.656,B 90.000,C 0.000} C_DIS
LIN {X 252.796,Y 142.107,Z 162.149,A -150.658,B 90.000,C 0.000} C_DIS
LIN {X 253.016,Y 141.714,Z 160.252,A -150.747,B 90.000,C 0.000} C_DIS
LIN {X 253.030,Y 141.689,Z 159.839,A -150.752,B 90.000,C 0.000} C_DIS
LIN {X 253.023,Y 141.701,Z 159.730,A -150.750,B 90.000,C 0.000} C_DIS
RET=EKI_SetBool("oxy","torchState",FALSE)
RET = EKI_Send("oxy","torchState")
PTP {X 251.278,Y 140.724,Z 159.730,A -150.750,B 90.000,C 0.000}
PTP {X 235.573,Y 131.929,Z 159.730,A -150.750,B 90.000,C 0.000}
PTP {X 240.417,Y 122.880,Z 164.140,A -152.928,B 90.000,C 0.000}
PTP {X 256.445,Y 131.072,Z 164.140,A -152.928,B 90.000,C 0.000}
WAIT SEC 2
RET=EKI_SetBool("oxy","torchState",TRUE)
RET = EKI_Send("oxy","torchState")
LIN {X 258.226,Y 131.982,Z 164.140,A -152.928,B 90.000,C 0.000} C_DIS
LIN {X 258.533,Y 131.379,Z 162.229,A -153.062,B 90.000,C 0.000} C_DIS
LIN {X 258.545,Y 131.357,Z 162.101,A -153.067,B 90.000,C 0.000} C_DIS
LIN {X 258.564,Y 131.320,Z 162.058,A -153.075,B 90.000,C 0.000} C_DIS
LIN {X 258.646,Y 131.158,Z 161.774,A -153.111,B 90.000,C 0.000} C_DIS
LIN {X 258.668,Y 131.114,Z 161.660,A -153.120,B 90.000,C 0.000} C_DIS
LIN {X 258.722,Y 131.007,Z 161.489,A -153.144,B 90.000,C 0.000} C_DIS
LIN {X 258.745,Y 130.962,Z 161.375,A -153.154,B 90.000,C 0.000} C_DIS
LIN {X 258.799,Y 130.854,Z 161.205,A -153.178,B 90.000,C 0.000} C_DIS
LIN {X 258.811,Y 130.832,Z 161.148,A -153.183,B 90.000,C 0.000} C_DIS
LIN {X 258.818,Y 130.817,Z 161.091,A -153.186,B 90.000,C 0.000} C_DIS
LIN {X 258.901,Y 130.654,Z 160.977,A -153.222,B 90.000,C 0.000} C_DIS
LIN {X 259.002,Y 130.453,Z 160.868,A -153.267,B 90.000,C 0.000} C_DIS
LIN {X 259.091,Y 130.277,Z 160.953,A -153.306,B 90.000,C 0.000} C_DIS
LIN {X 259.171,Y 130.116,Z 161.246,A -153.341,B 90.000,C 0.000} C_DIS
LIN {X 259.200,Y 130.059,Z 161.477,A -153.354,B 90.000,C 0.000} C_DIS
LIN {X 259.231,Y 129.998,Z 163.975,A -153.367,B 90.000,C 0.000} C_DIS
LIN {X 259.208,Y 130.043,Z 165.166,A -153.357,B 90.000,C 0.000} C_DIS
LIN {X 259.039,Y 130.380,Z 166.781,A -153.283,B 90.000,C 0.000} C_DIS
LIN {X 259.000,Y 130.458,Z 166.985,A -153.266,B 90.000,C 0.000} C_DIS
LIN {X 258.995,Y 130.467,Z 167.085,A -153.264,B 90.000,C 0.000} C_DIS
LIN {X 258.983,Y 130.490,Z 167.122,A -153.258,B 90.000,C 0.000} C_DIS
LIN {X 258.965,Y 130.527,Z 167.236,A -153.250,B 90.000,C 0.000} C_DIS
LIN {X 258.955,Y 130.546,Z 167.350,A -153.246,B 90.000,C 0.000} C_DIS
LIN {X 258.821,Y 130.811,Z 168.146,A -153.187,B 90.000,C 0.000} C_DIS
LIN {X 258.790,Y 130.874,Z 168.507,A -153.174,B 90.000,C 0.000} C_DIS
LIN {X 258.777,Y 130.899,Z 168.544,A -153.168,B 90.000,C 0.000} C_DIS
LIN {X 258.652,Y 131.145,Z 169.094,A -153.113,B 90.000,C 0.000} C_DIS
LIN {X 258.648,Y 131.153,Z 169.193,A -153.112,B 90.000,C 0.000} C_DIS
LIN {X 258.539,Y 131.368,Z 169.739,A -153.064,B 90.000,C 0.000} C_DIS
LIN {X 258.522,Y 131.401,Z 169.967,A -153.057,B 90.000,C 0.000} C_DIS
LIN {X 258.408,Y 131.625,Z 170.422,A -153.007,B 90.000,C 0.000} C_DIS
LIN {X 258.402,Y 131.637,Z 170.506,A -153.004,B 90.000,C 0.000} C_DIS
LIN {X 258.375,Y 131.689,Z 170.681,A -152.993,B 90.000,C 0.000} C_DIS
LIN {X 258.334,Y 131.770,Z 170.853,A -152.975,B 90.000,C 0.000} C_DIS
LIN {X 258.308,Y 131.821,Z 170.934,A -152.964,B 90.000,C 0.000} C_DIS
LIN {X 258.287,Y 131.864,Z 170.977,A -152.954,B 90.000,C 0.000} C_DIS
LIN {X 258.074,Y 132.279,Z 172.015,A -152.862,B 90.000,C 0.000} C_DIS
LIN {X 258.064,Y 132.300,Z 172.143,A -152.857,B 90.000,C 0.000} C_DIS
LIN {X 258.050,Y 132.327,Z 172.243,A -152.851,B 90.000,C 0.000} C_DIS
LIN {X 257.945,Y 132.530,Z 172.608,A -152.806,B 90.000,C 0.000} C_DIS
LIN {X 257.878,Y 132.662,Z 172.868,A -152.777,B 90.000,C 0.000} C_DIS
LIN {X 257.711,Y 132.985,Z 173.594,A -152.705,B 90.000,C 0.000} C_DIS
LIN {X 257.602,Y 133.196,Z 173.949,A -152.658,B 90.000,C 0.000} C_DIS
LIN {X 257.582,Y 133.235,Z 174.063,A -152.650,B 90.000,C 0.000} C_DIS
LIN {X 257.554,Y 133.289,Z 174.145,A -152.638,B 90.000,C 0.000} C_DIS
LIN {X 257.514,Y 133.366,Z 174.313,A -152.620,B 90.000,C 0.000} C_DIS
LIN {X 257.338,Y 133.705,Z 174.917,A -152.545,B 90.000,C 0.000} C_DIS
LIN {X 257.332,Y 133.718,Z 174.974,A -152.542,B 90.000,C 0.000} C_DIS
LIN {X 257.320,Y 133.740,Z 175.031,A -152.537,B 90.000,C 0.000} C_DIS
LIN {X 257.292,Y 133.794,Z 175.112,A -152.525,B 90.000,C 0.000} C_DIS
LIN {X 257.202,Y 133.967,Z 175.474,A -152.487,B 90.000,C 0.000} C_DIS
LIN {X 257.029,Y 134.298,Z 176.092,A -152.413,B 90.000,C 0.000} C_DIS
LIN {X 257.001,Y 134.352,Z 176.168,A -152.401,B 90.000,C 0.000} C_DIS
LIN {X 256.978,Y 134.396,Z 176.282,A -152.391,B 90.000,C 0.000} C_DIS
LIN {X 256.922,Y 134.503,Z 176.453,A -152.367,B 90.000,C 0.000} C_DIS
LIN {X 256.909,Y 134.527,Z 176.506,A -152.362,B 90.000,C 0.000} C_DIS
LIN {X 256.832,Y 134.674,Z 176.685,A -152.329,B 90.000,C 0.000} C_DIS
LIN {X 256.822,Y 134.693,Z 176.737,A -152.325,B 90.000,C 0.000} C_DIS
LIN {X 256.157,Y 135.954,Z 178.791,A -152.043,B 90.000,C 0.000} C_DIS
LIN {X 255.914,Y 136.412,Z 179.466,A -151.941,B 90.000,C 0.000} C_DIS
LIN {X 255.883,Y 136.470,Z 179.525,A -151.928,B 90.000,C 0.000} C_DIS
LIN {X 255.869,Y 136.496,Z 179.562,A -151.922,B 90.000,C 0.000} C_DIS
LIN {X 255.820,Y 136.588,Z 179.730,A -151.901,B 90.000,C 0.000} C_DIS
LIN {X 255.753,Y 136.713,Z 179.896,A -151.873,B 90.000,C 0.000} C_DIS
LIN {X 255.720,Y 136.775,Z 180.011,A -151.859,B 90.000,C 0.000} C_DIS
LIN {X 255.107,Y 137.915,Z 181.573,A -151.604,B 90.000,C 0.000} C_DIS
LIN {X 255.058,Y 138.005,Z 181.662,A -151.583,B 90.000,C 0.000} C_DIS
LIN {X 254.345,Y 139.315,Z 183.399,A -151.289,B 90.000,C 0.000} C_DIS
LIN {X 254.246,Y 139.495,Z 183.549,A -151.248,B 90.000,C 0.000} C_DIS
LIN {X 254.145,Y 139.679,Z 183.825,A -151.207,B 90.000,C 0.000} C_DIS
LIN {X 253.940,Y 140.051,Z 184.273,A -151.123,B 90.000,C 0.000} C_DIS
LIN {X 253.825,Y 140.260,Z 184.475,A -151.076,B 90.000,C 0.000} C_DIS
LIN {X 253.783,Y 140.336,Z 184.586,A -151.058,B 90.000,C 0.000} C_DIS
LIN {X 253.629,Y 140.613,Z 184.903,A -150.996,B 90.000,C 0.000} C_DIS
LIN {X 253.585,Y 140.694,Z 184.968,A -150.978,B 90.000,C 0.000} C_DIS
LIN {X 253.381,Y 141.060,Z 185.386,A -150.895,B 90.000,C 0.000} C_DIS
LIN {X 253.355,Y 141.108,Z 185.471,A -150.884,B 90.000,C 0.000} C_DIS
LIN {X 253.313,Y 141.182,Z 185.556,A -150.867,B 90.000,C 0.000} C_DIS
LIN {X 253.272,Y 141.257,Z 185.604,A -150.850,B 90.000,C 0.000} C_DIS
LIN {X 253.047,Y 141.659,Z 186.068,A -150.759,B 90.000,C 0.000} C_DIS
LIN {X 253.023,Y 141.701,Z 186.182,A -150.750,B 90.000,C 0.000} C_DIS
LIN {X 252.262,Y 143.052,Z 187.548,A -150.444,B 90.000,C 0.000} C_DIS
LIN {X 252.243,Y 143.085,Z 187.661,A -150.436,B 90.000,C 0.000} C_DIS
LIN {X 251.981,Y 143.547,Z 188.060,A -150.331,B 90.000,C 0.000} C_DIS
LIN {X 251.963,Y 143.579,Z 188.173,A -150.324,B 90.000,C 0.000} C_DIS
LIN {X 251.501,Y 144.386,Z 188.913,A -150.140,B 90.000,C 0.000} C_DIS
LIN {X 251.492,Y 144.401,Z 188.970,A -150.137,B 90.000,C 0.000} C_DIS
LIN {X 251.471,Y 144.437,Z 189.027,A -150.128,B 90.000,C 0.000} C_DIS
LIN {X 250.675,Y 145.815,Z 190.279,A -149.814,B 90.000,C 0.000} C_DIS
LIN {X 250.664,Y 145.834,Z 190.327,A -149.810,B 90.000,C 0.000} C_DIS
LIN {X 250.538,Y 146.051,Z 190.562,A -149.760,B 90.000,C 0.000} C_DIS
LIN {X 250.276,Y 146.500,Z 190.961,A -149.657,B 90.000,C 0.000} C_DIS
LIN {X 250.196,Y 146.636,Z 191.046,A -149.626,B 90.000,C 0.000} C_DIS
LIN {X 249.230,Y 148.272,Z 192.540,A -149.251,B 90.000,C 0.000} C_DIS
LIN {X 249.163,Y 148.383,Z 192.611,A -149.225,B 90.000,C 0.000} C_DIS
LIN {X 248.900,Y 148.825,Z 192.978,A -149.124,B 90.000,C 0.000} C_DIS
LIN {X 248.846,Y 148.916,Z 193.068,A -149.103,B 90.000,C 0.000} C_DIS
LIN {X 248.837,Y 148.931,Z 193.123,A -149.099,B 90.000,C 0.000} C_DIS
LIN {X 248.636,Y 149.266,Z 193.351,A -149.022,B 90.000,C 0.000} C_DIS
LIN {X 248.437,Y 149.597,Z 193.641,A -148.946,B 90.000,C 0.000} C_DIS
LIN {X 248.427,Y 149.614,Z 193.692,A -148.942,B 90.000,C 0.000} C_DIS
LIN {X 248.225,Y 149.948,Z 193.920,A -148.865,B 90.000,C 0.000} C_DIS
LIN {X 247.821,Y 150.614,Z 194.489,A -148.711,B 90.000,C 0.000} C_DIS
LIN {X 247.719,Y 150.782,Z 194.588,A -148.672,B 90.000,C 0.000} C_DIS
LIN {X 246.657,Y 152.513,Z 195.969,A -148.271,B 90.000,C 0.000} C_DIS
LIN {X 245.531,Y 154.320,Z 197.279,A -147.850,B 90.000,C 0.000} C_DIS
LIN {X 245.478,Y 154.404,Z 197.334,A -147.830,B 90.000,C 0.000} C_DIS
LIN {X 245.437,Y 154.469,Z 197.394,A -147.815,B 90.000,C 0.000} C_DIS
LIN {X 245.377,Y 154.565,Z 197.443,A -147.793,B 90.000,C 0.000} C_DIS
LIN {X 244.221,Y 156.384,Z 198.710,A -147.367,B 90.000,C 0.000} C_DIS
LIN {X 243.033,Y 158.224,Z 199.915,A -146.934,B 90.000,C 0.000} C_DIS
LIN {X 241.810,Y 160.087,Z 201.048,A -146.494,B 90.000,C 0.000} C_DIS
LIN {X 240.554,Y 161.969,Z 202.112,A -146.047,B 90.000,C 0.000} C_DIS
LIN {X 239.264,Y 163.868,Z 203.100,A -145.593,B 90.000,C 0.000} C_DIS
LIN {X 237.932,Y 165.796,Z 203.972,A -145.130,B 90.000,C 0.000} C_DIS
LIN {X 237.833,Y 165.939,Z 204.034,A -145.096,B 90.000,C 0.000} C_DIS
LIN {X 237.713,Y 166.109,Z 204.145,A -145.055,B 90.000,C 0.000} C_DIS
LIN {X 237.620,Y 166.243,Z 204.173,A -145.023,B 90.000,C 0.000} C_DIS
LIN {X 237.549,Y 166.345,Z 204.083,A -144.998,B 90.000,C 0.000} C_DIS
LIN {X 236.892,Y 167.278,Z 201.859,A -144.773,B 90.000,C 0.000} C_DIS
LIN {X 236.291,Y 168.127,Z 199.586,A -144.567,B 90.000,C 0.000} C_DIS
LIN {X 235.719,Y 168.928,Z 197.288,A -144.373,B 90.000,C 0.000} C_DIS
LIN {X 235.187,Y 169.668,Z 194.960,A -144.193,B 90.000,C 0.000} C_DIS
LIN {X 234.817,Y 170.179,Z 193.224,A -144.068,B 90.000,C 0.000} C_DIS
LIN {X 234.808,Y 170.191,Z 193.137,A -144.065,B 90.000,C 0.000} C_DIS
LIN {X 234.342,Y 170.833,Z 190.766,A -143.908,B 90.000,C 0.000} C_DIS
LIN {X 233.992,Y 171.312,Z 188.749,A -143.791,B 90.000,C 0.000} C_DIS
LIN {X 233.965,Y 171.348,Z 188.692,A -143.782,B 90.000,C 0.000} C_DIS
LIN {X 233.564,Y 171.894,Z 186.285,A -143.648,B 90.000,C 0.000} C_DIS
LIN {X 233.206,Y 172.380,Z 183.860,A -143.529,B 90.000,C 0.000} C_DIS
LIN {X 232.877,Y 172.824,Z 181.422,A -143.420,B 90.000,C 0.000} C_DIS
LIN {X 232.794,Y 172.936,Z 180.666,A -143.392,B 90.000,C 0.000} C_DIS
LIN {X 232.800,Y 172.928,Z 180.606,A -143.394,B 90.000,C 0.000} C_DIS
LIN {X 233.285,Y 172.273,Z 181.232,A -143.555,B 90.000,C 0.000} C_DIS
LIN {X 233.318,Y 172.229,Z 181.299,A -143.566,B 90.000,C 0.000} C_DIS
LIN {X 233.338,Y 172.202,Z 181.331,A -143.573,B 90.000,C 0.000} C_DIS
LIN {X 233.549,Y 171.915,Z 181.574,A -143.643,B 90.000,C 0.000} C_DIS
LIN {X 233.588,Y 171.863,Z 181.640,A -143.656,B 90.000,C 0.000} C_DIS
LIN {X 233.609,Y 171.833,Z 181.669,A -143.663,B 90.000,C 0.000} C_DIS
LIN {X 234.428,Y 170.715,Z 182.662,A -143.937,B 90.000,C 0.000} C_DIS
LIN {X 234.642,Y 170.421,Z 182.841,A -144.009,B 90.000,C 0.000} C_DIS
LIN {X 234.762,Y 170.255,Z 182.999,A -144.050,B 90.000,C 0.000} C_DIS
LIN {X 234.829,Y 170.163,Z 183.047,A -144.072,B 90.000,C 0.000} C_DIS
LIN {X 235.758,Y 168.874,Z 184.006,A -144.386,B 90.000,C 0.000} C_DIS
LIN {X 235.792,Y 168.825,Z 184.061,A -144.398,B 90.000,C 0.000} C_DIS
LIN {X 236.033,Y 168.488,Z 184.202,A -144.479,B 90.000,C 0.000} C_DIS
LIN {X 236.058,Y 168.454,Z 184.248,A -144.488,B 90.000,C 0.000} C_DIS
LIN {X 236.105,Y 168.387,Z 184.305,A -144.504,B 90.000,C 0.000} C_DIS
LIN {X 236.210,Y 168.240,Z 184.404,A -144.540,B 90.000,C 0.000} C_DIS
LIN {X 236.270,Y 168.156,Z 184.484,A -144.560,B 90.000,C 0.000} C_DIS
LIN {X 236.777,Y 167.441,Z 184.888,A -144.733,B 90.000,C 0.000} C_DIS
LIN {X 236.819,Y 167.383,Z 184.899,A -144.747,B 90.000,C 0.000} C_DIS
LIN {X 236.849,Y 167.340,Z 184.918,A -144.758,B 90.000,C 0.000} C_DIS
LIN {X 236.890,Y 167.282,Z 184.970,A -144.772,B 90.000,C 0.000} C_DIS
LIN {X 238.219,Y 165.383,Z 185.844,A -145.230,B 90.000,C 0.000} C_DIS
LIN {X 238.284,Y 165.289,Z 185.857,A -145.252,B 90.000,C 0.000} C_DIS
LIN {X 238.414,Y 165.102,Z 185.938,A -145.297,B 90.000,C 0.000} C_DIS
LIN {X 238.464,Y 165.030,Z 185.951,A -145.315,B 90.000,C 0.000} C_DIS
LIN {X 239.834,Y 163.032,Z 186.565,A -145.793,B 90.000,C 0.000} C_DIS
LIN {X 239.956,Y 162.853,Z 186.611,A -145.836,B 90.000,C 0.000} C_DIS
LIN {X 239.990,Y 162.803,Z 186.640,A -145.848,B 90.000,C 0.000} C_DIS
LIN {X 240.150,Y 162.567,Z 186.696,A -145.904,B 90.000,C 0.000} C_DIS
LIN {X 240.178,Y 162.525,Z 186.726,A -145.914,B 90.000,C 0.000} C_DIS
LIN {X 241.150,Y 161.080,Z 186.924,A -146.258,B 90.000,C 0.000} C_DIS
LIN {X 242.328,Y 159.302,Z 186.922,A -146.680,B 90.000,C 0.000} C_DIS
LIN {X 242.399,Y 159.195,Z 186.943,A -146.705,B 90.000,C 0.000} C_DIS
LIN {X 243.759,Y 157.104,Z 186.775,A -147.198,B 90.000,C 0.000} C_DIS
LIN {X 245.095,Y 155.011,Z 186.484,A -147.689,B 90.000,C 0.000} C_DIS
LIN {X 246.404,Y 152.922,Z 186.067,A -148.176,B 90.000,C 0.000} C_DIS
LIN {X 247.698,Y 150.813,Z 185.714,A -148.665,B 90.000,C 0.000} C_DIS
LIN {X 248.967,Y 148.709,Z 185.254,A -149.150,B 90.000,C 0.000} C_DIS
LIN {X 249.598,Y 147.651,Z 184.942,A -149.393,B 90.000,C 0.000} C_DIS
LIN {X 249.642,Y 147.577,Z 184.884,A -149.410,B 90.000,C 0.000} C_DIS
LIN {X 250.811,Y 145.582,Z 183.935,A -149.867,B 90.000,C 0.000} C_DIS
LIN {X 251.900,Y 143.689,Z 182.718,A -150.299,B 90.000,C 0.000} C_DIS
LIN {X 251.940,Y 143.618,Z 182.655,A -150.315,B 90.000,C 0.000} C_DIS
LIN {X 252.146,Y 143.256,Z 182.427,A -150.397,B 90.000,C 0.000} C_DIS
LIN {X 252.677,Y 142.318,Z 181.662,A -150.610,B 90.000,C 0.000} C_DIS
LIN {X 252.729,Y 142.226,Z 181.572,A -150.631,B 90.000,C 0.000} C_DIS
LIN {X 252.736,Y 142.213,Z 181.517,A -150.634,B 90.000,C 0.000} C_DIS
LIN {X 253.019,Y 141.709,Z 181.118,A -150.748,B 90.000,C 0.000} C_DIS
LIN {X 253.915,Y 140.096,Z 179.432,A -151.113,B 90.000,C 0.000} C_DIS
LIN {X 254.164,Y 139.645,Z 178.884,A -151.214,B 90.000,C 0.000} C_DIS
LIN {X 254.207,Y 139.567,Z 178.815,A -151.232,B 90.000,C 0.000} C_DIS
LIN {X 254.469,Y 139.088,Z 178.278,A -151.340,B 90.000,C 0.000} C_DIS
LIN {X 255.224,Y 137.698,Z 176.342,A -151.652,B 90.000,C 0.000} C_DIS
LIN {X 255.404,Y 137.365,Z 175.835,A -151.727,B 90.000,C 0.000} C_DIS
LIN {X 255.435,Y 137.306,Z 175.770,A -151.740,B 90.000,C 0.000} C_DIS
LIN {X 255.449,Y 137.280,Z 175.733,A -151.746,B 90.000,C 0.000} C_DIS
LIN {X 255.565,Y 137.064,Z 175.375,A -151.795,B 90.000,C 0.000} C_DIS
LIN {X 255.612,Y 136.976,Z 175.282,A -151.814,B 90.000,C 0.000} C_DIS
LIN {X 255.641,Y 136.922,Z 175.138,A -151.826,B 90.000,C 0.000} C_DIS
LIN {X 255.684,Y 136.842,Z 174.986,A -151.844,B 90.000,C 0.000} C_DIS
LIN {X 255.902,Y 136.433,Z 174.334,A -151.936,B 90.000,C 0.000} C_DIS
LIN {X 255.940,Y 136.363,Z 174.177,A -151.952,B 90.000,C 0.000} C_DIS
LIN {X 256.130,Y 136.005,Z 173.608,A -152.032,B 90.000,C 0.000} C_DIS
LIN {X 256.154,Y 135.959,Z 173.523,A -152.042,B 90.000,C 0.000} C_DIS
LIN {X 256.200,Y 135.873,Z 173.403,A -152.061,B 90.000,C 0.000} C_DIS
LIN {X 256.284,Y 135.715,Z 173.039,A -152.097,B 90.000,C 0.000} C_DIS
LIN {X 256.329,Y 135.629,Z 172.914,A -152.116,B 90.000,C 0.000} C_DIS
LIN {X 256.421,Y 135.457,Z 172.551,A -152.154,B 90.000,C 0.000} C_DIS
LIN {X 256.449,Y 135.403,Z 172.470,A -152.166,B 90.000,C 0.000} C_DIS
LIN {X 256.472,Y 135.359,Z 172.356,A -152.176,B 90.000,C 0.000} C_DIS
LIN {X 256.528,Y 135.252,Z 172.186,A -152.200,B 90.000,C 0.000} C_DIS
LIN {X 256.550,Y 135.211,Z 172.072,A -152.209,B 90.000,C 0.000} C_DIS
LIN {X 256.595,Y 135.126,Z 171.947,A -152.228,B 90.000,C 0.000} C_DIS
LIN {X 256.686,Y 134.953,Z 171.584,A -152.267,B 90.000,C 0.000} C_DIS
LIN {X 256.714,Y 134.900,Z 171.503,A -152.279,B 90.000,C 0.000} C_DIS
LIN {X 256.727,Y 134.875,Z 171.451,A -152.284,B 90.000,C 0.000} C_DIS
LIN {X 256.732,Y 134.866,Z 171.380,A -152.286,B 90.000,C 0.000} C_DIS
LIN {X 256.897,Y 134.550,Z 170.663,A -152.357,B 90.000,C 0.000} C_DIS
LIN {X 257.082,Y 134.197,Z 169.934,A -152.435,B 90.000,C 0.000} C_DIS
LIN {X 257.110,Y 134.144,Z 169.853,A -152.447,B 90.000,C 0.000} C_DIS
LIN {X 257.218,Y 133.937,Z 169.341,A -152.493,B 90.000,C 0.000} C_DIS
LIN {X 257.232,Y 133.909,Z 169.227,A -152.500,B 90.000,C 0.000} C_DIS
LIN {X 257.322,Y 133.737,Z 168.815,A -152.538,B 90.000,C 0.000} C_DIS
LIN {X 257.344,Y 133.693,Z 168.772,A -152.548,B 90.000,C 0.000} C_DIS
LIN {X 257.453,Y 133.485,Z 168.260,A -152.594,B 90.000,C 0.000} C_DIS
LIN {X 257.540,Y 133.316,Z 167.919,A -152.631,B 90.000,C 0.000} C_DIS
LIN {X 257.546,Y 133.304,Z 167.847,A -152.634,B 90.000,C 0.000} C_DIS
LIN {X 257.663,Y 133.078,Z 167.293,A -152.684,B 90.000,C 0.000} C_DIS
LIN {X 257.681,Y 133.044,Z 167.250,A -152.692,B 90.000,C 0.000} C_DIS
LIN {X 257.844,Y 132.727,Z 166.311,A -152.762,B 90.000,C 0.000} C_DIS
LIN {X 257.897,Y 132.624,Z 166.098,A -152.785,B 90.000,C 0.000} C_DIS
LIN {X 257.906,Y 132.606,Z 165.984,A -152.789,B 90.000,C 0.000} C_DIS
LIN {X 257.922,Y 132.575,Z 165.870,A -152.796,B 90.000,C 0.000} C_DIS
LIN {X 257.933,Y 132.553,Z 165.817,A -152.801,B 90.000,C 0.000} C_DIS
LIN {X 257.945,Y 132.531,Z 165.729,A -152.806,B 90.000,C 0.000} C_DIS
LIN {X 258.054,Y 132.319,Z 165.188,A -152.853,B 90.000,C 0.000} C_DIS
LIN {X 258.068,Y 132.291,Z 165.074,A -152.859,B 90.000,C 0.000} C_DIS
LIN {X 258.222,Y 131.990,Z 164.240,A -152.926,B 90.000,C 0.000} C_DIS
LIN {X 258.226,Y 131.982,Z 164.140,A -152.928,B 90.000,C 0.000} C_DIS
RET=EKI_SetBool("oxy","torchState",FALSE)
RET = EKI_Send("oxy","torchState")
PTP {X 256.445,Y 131.072,Z 164.140,A -152.928,B 90.000,C 0.000}
PTP {X 240.417,Y 122.880,Z 164.140,A -152.928,B 90.000,C 0.000}
PTP {X 242.252,Y 119.223,Z 164.405,A -153.796,B 90.000,C 0.000}
PTP {X 258.402,Y 127.171,Z 164.405,A -153.796,B 90.000,C 0.000}
WAIT SEC 2
RET=EKI_SetBool("oxy","torchState",TRUE)
RET = EKI_Send("oxy","torchState")
LIN {X 260.196,Y 128.054,Z 164.405,A -153.796,B 90.000,C 0.000} C_DIS
LIN {X 260.322,Y 127.798,Z 163.481,A -153.852,B 90.000,C 0.000} C_DIS
LIN {X 260.543,Y 127.347,Z 161.617,A -153.952,B 90.000,C 0.000} C_DIS
LIN {X 260.554,Y 127.325,Z 161.432,A -153.957,B 90.000,C 0.000} C_DIS
LIN {X 260.844,Y 126.730,Z 159.022,A -154.087,B 90.000,C 0.000} C_DIS
LIN {X 260.908,Y 126.598,Z 158.592,A -154.116,B 90.000,C 0.000} C_DIS
LIN {X 260.998,Y 126.413,Z 157.606,A -154.157,B 90.000,C 0.000} C_DIS
LIN {X 261.015,Y 126.378,Z 157.507,A -154.165,B 90.000,C 0.000} C_DIS
LIN {X 261.111,Y 126.179,Z 156.770,A -154.208,B 90.000,C 0.000} C_DIS
LIN {X 261.118,Y 126.164,Z 156.642,A -154.212,B 90.000,C 0.000} C_DIS
LIN {X 261.397,Y 125.585,Z 154.226,A -154.338,B 90.000,C 0.000} C_DIS
LIN {X 261.555,Y 125.255,Z 152.854,A -154.411,B 90.000,C 0.000} C_DIS
LIN {X 261.596,Y 125.169,Z 152.730,A -154.430,B 90.000,C 0.000} C_DIS
LIN {X 261.656,Y 125.044,Z 153.158,A -154.457,B 90.000,C 0.000} C_DIS
LIN {X 261.827,Y 124.686,Z 155.627,A -154.535,B 90.000,C 0.000} C_DIS
LIN {X 262.012,Y 124.298,Z 158.089,A -154.620,B 90.000,C 0.000} C_DIS
LIN {X 262.171,Y 123.961,Z 160.561,A -154.694,B 90.000,C 0.000} C_DIS
LIN {X 262.342,Y 123.598,Z 163.029,A -154.773,B 90.000,C 0.000} C_DIS
LIN {X 262.514,Y 123.234,Z 165.496,A -154.853,B 90.000,C 0.000} C_DIS
LIN {X 262.683,Y 122.872,Z 167.964,A -154.932,B 90.000,C 0.000} C_DIS
LIN {X 262.856,Y 122.502,Z 170.430,A -155.013,B 90.000,C 0.000} C_DIS
LIN {X 263.014,Y 122.162,Z 172.783,A -155.087,B 90.000,C 0.000} C_DIS
LIN {X 263.342,Y 121.453,Z 175.158,A -155.241,B 90.000,C 0.000} C_DIS
LIN {X 263.495,Y 121.122,Z 176.141,A -155.313,B 90.000,C 0.000} C_DIS
LIN {X 263.537,Y 121.029,Z 176.327,A -155.333,B 90.000,C 0.000} C_DIS
LIN {X 263.602,Y 120.888,Z 176.866,A -155.364,B 90.000,C 0.000} C_DIS
LIN {X 264.002,Y 120.013,Z 179.173,A -155.554,B 90.000,C 0.000} C_DIS
LIN {X 264.415,Y 119.099,Z 181.463,A -155.752,B 90.000,C 0.000} C_DIS
LIN {X 264.854,Y 118.121,Z 183.722,A -155.964,B 90.000,C 0.000} C_DIS
LIN {X 265.311,Y 117.090,Z 185.953,A -156.187,B 90.000,C 0.000} C_DIS
LIN {X 265.786,Y 116.007,Z 188.155,A -156.420,B 90.000,C 0.000} C_DIS
LIN {X 265.844,Y 115.875,Z 188.458,A -156.449,B 90.000,C 0.000} C_DIS
LIN {X 265.953,Y 115.625,Z 188.878,A -156.503,B 90.000,C 0.000} C_DIS
LIN {X 266.026,Y 115.456,Z 189.255,A -156.539,B 90.000,C 0.000} C_DIS
LIN {X 266.082,Y 115.328,Z 189.439,A -156.567,B 90.000,C 0.000} C_DIS
LIN {X 266.509,Y 114.337,Z 191.345,A -156.780,B 90.000,C 0.000} C_DIS
LIN {X 266.564,Y 114.209,Z 191.530,A -156.807,B 90.000,C 0.000} C_DIS
LIN {X 266.834,Y 113.578,Z 192.631,A -156.943,B 90.000,C 0.000} C_DIS
LIN {X 267.011,Y 113.159,Z 193.439,A -157.033,B 90.000,C 0.000} C_DIS
LIN {X 267.078,Y 113.001,Z 193.653,A -157.067,B 90.000,C 0.000} C_DIS
LIN {X 267.167,Y 112.792,Z 194.071,A -157.112,B 90.000,C 0.000} C_DIS
LIN {X 267.313,Y 112.445,Z 194.580,A -157.186,B 90.000,C 0.000} C_DIS
LIN {X 267.363,Y 112.325,Z 194.832,A -157.212,B 90.000,C 0.000} C_DIS
LIN {X 267.475,Y 112.058,Z 195.263,A -157.269,B 90.000,C 0.000} C_DIS
LIN {X 267.541,Y 111.900,Z 195.474,A -157.303,B 90.000,C 0.000} C_DIS
LIN {X 267.629,Y 111.690,Z 195.892,A -157.348,B 90.000,C 0.000} C_DIS
LIN {X 267.889,Y 111.065,Z 196.822,A -157.481,B 90.000,C 0.000} C_DIS
LIN {X 267.957,Y 110.902,Z 197.134,A -157.516,B 90.000,C 0.000} C_DIS
LIN {X 267.989,Y 110.823,Z 197.219,A -157.533,B 90.000,C 0.000} C_DIS
LIN {X 268.109,Y 110.532,Z 197.645,A -157.595,B 90.000,C 0.000} C_DIS
LIN {X 268.174,Y 110.376,Z 197.931,A -157.629,B 90.000,C 0.000} C_DIS
LIN {X 268.241,Y 110.212,Z 198.130,A -157.664,B 90.000,C 0.000} C_DIS
LIN {X 268.256,Y 110.175,Z 198.244,A -157.672,B 90.000,C 0.000} C_DIS
LIN {X 268.289,Y 110.096,Z 198.364,A -157.688,B 90.000,C 0.000} C_DIS
LIN {X 268.322,Y 110.016,Z 198.448,A -157.706,B 90.000,C 0.000} C_DIS
LIN {X 268.391,Y 109.845,Z 198.725,A -157.742,B 90.000,C 0.000} C_DIS
LIN {X 268.411,Y 109.797,Z 198.744,A -157.752,B 90.000,C 0.000} C_DIS
LIN {X 268.497,Y 109.586,Z 199.135,A -157.797,B 90.000,C 0.000} C_DIS
LIN {X 268.562,Y 109.428,Z 199.288,A -157.831,B 90.000,C 0.000} C_DIS
LIN {X 268.599,Y 109.336,Z 199.482,A -157.851,B 90.000,C 0.000} C_DIS
LIN {X 268.739,Y 108.994,Z 199.960,A -157.924,B 90.000,C 0.000} C_DIS
LIN {X 268.776,Y 108.901,Z 200.123,A -157.943,B 90.000,C 0.000} C_DIS
LIN {X 268.840,Y 108.743,Z 200.298,A -157.977,B 90.000,C 0.000} C_DIS
LIN {X 269.079,Y 108.149,Z 201.139,A -158.104,B 90.000,C 0.000} C_DIS
LIN {X 269.116,Y 108.057,Z 201.301,A -158.123,B 90.000,C 0.000} C_DIS
LIN {X 269.254,Y 107.713,Z 201.772,A -158.196,B 90.000,C 0.000} C_DIS
LIN {X 269.307,Y 107.582,Z 201.898,A -158.224,B 90.000,C 0.000} C_DIS
LIN {X 269.344,Y 107.489,Z 202.065,A -158.244,B 90.000,C 0.000} C_DIS
LIN {X 269.795,Y 106.352,Z 203.539,A -158.486,B 90.000,C 0.000} C_DIS
LIN {X 269.831,Y 106.259,Z 203.708,A -158.505,B 90.000,C 0.000} C_DIS
LIN {X 269.894,Y 106.101,Z 203.911,A -158.539,B 90.000,C 0.000} C_DIS
LIN {X 269.956,Y 105.942,Z 204.070,A -158.573,B 90.000,C 0.000} C_DIS
LIN {X 270.018,Y 105.783,Z 204.302,A -158.607,B 90.000,C 0.000} C_DIS
LIN {X 270.050,Y 105.703,Z 204.389,A -158.624,B 90.000,C 0.000} C_DIS
LIN {X 270.081,Y 105.624,Z 204.446,A -158.640,B 90.000,C 0.000} C_DIS
LIN {X 270.668,Y 104.111,Z 206.347,A -158.961,B 90.000,C 0.000} C_DIS
LIN {X 270.698,Y 104.032,Z 206.443,A -158.978,B 90.000,C 0.000} C_DIS
LIN {X 270.739,Y 103.926,Z 206.484,A -159.000,B 90.000,C 0.000} C_DIS
LIN {X 270.942,Y 103.395,Z 207.193,A -159.113,B 90.000,C 0.000} C_DIS
LIN {X 271.306,Y 102.435,Z 208.144,A -159.315,B 90.000,C 0.000} C_DIS
LIN {X 271.332,Y 102.367,Z 208.264,A -159.330,B 90.000,C 0.000} C_DIS
LIN {X 271.364,Y 102.281,Z 208.345,A -159.348,B 90.000,C 0.000} C_DIS
LIN {X 271.386,Y 102.224,Z 208.374,A -159.360,B 90.000,C 0.000} C_DIS
LIN {X 271.707,Y 101.368,Z 209.282,A -159.540,B 90.000,C 0.000} C_DIS
LIN {X 271.725,Y 101.319,Z 209.367,A -159.551,B 90.000,C 0.000} C_DIS
LIN {X 271.785,Y 101.159,Z 209.538,A -159.585,B 90.000,C 0.000} C_DIS
LIN {X 271.802,Y 101.113,Z 209.623,A -159.594,B 90.000,C 0.000} C_DIS
LIN {X 272.244,Y 99.915,Z 210.725,A -159.847,B 90.000,C 0.000} C_DIS
LIN {X 272.296,Y 99.773,Z 210.932,A -159.877,B 90.000,C 0.000} C_DIS
LIN {X 272.878,Y 98.171,Z 212.354,A -160.213,B 90.000,C 0.000} C_DIS
LIN {X 272.899,Y 98.113,Z 212.415,A -160.225,B 90.000,C 0.000} C_DIS
LIN {X 272.917,Y 98.063,Z 212.442,A -160.236,B 90.000,C 0.000} C_DIS
LIN {X 272.977,Y 97.895,Z 212.608,A -160.271,B 90.000,C 0.000} C_DIS
LIN {X 272.995,Y 97.845,Z 212.635,A -160.282,B 90.000,C 0.000} C_DIS
LIN {X 273.016,Y 97.788,Z 212.696,A -160.294,B 90.000,C 0.000} C_DIS
LIN {X 273.327,Y 96.913,Z 213.394,A -160.477,B 90.000,C 0.000} C_DIS
LIN {X 273.359,Y 96.825,Z 213.492,A -160.496,B 90.000,C 0.000} C_DIS
LIN {X 273.478,Y 96.486,Z 213.738,A -160.567,B 90.000,C 0.000} C_DIS
LIN {X 273.491,Y 96.452,Z 213.767,A -160.574,B 90.000,C 0.000} C_DIS
LIN {X 273.510,Y 96.395,Z 213.834,A -160.586,B 90.000,C 0.000} C_DIS
LIN {X 274.179,Y 94.477,Z 215.290,A -160.987,B 90.000,C 0.000} C_DIS
LIN {X 274.325,Y 94.052,Z 215.540,A -161.076,B 90.000,C 0.000} C_DIS
LIN {X 274.350,Y 93.979,Z 215.601,A -161.091,B 90.000,C 0.000} C_DIS
LIN {X 274.387,Y 93.872,Z 215.646,A -161.113,B 90.000,C 0.000} C_DIS
LIN {X 274.456,Y 93.670,Z 215.832,A -161.156,B 90.000,C 0.000} C_DIS
LIN {X 274.534,Y 93.441,Z 215.999,A -161.203,B 90.000,C 0.000} C_DIS
LIN {X 274.584,Y 93.293,Z 216.077,A -161.234,B 90.000,C 0.000} C_DIS
LIN {X 275.091,Y 91.789,Z 216.992,A -161.548,B 90.000,C 0.000} C_DIS
LIN {X 275.100,Y 91.760,Z 217.105,A -161.554,B 90.000,C 0.000} C_DIS
LIN {X 274.625,Y 93.172,Z 218.787,A -161.260,B 90.000,C 0.000} C_DIS
LIN {X 274.570,Y 93.333,Z 218.895,A -161.226,B 90.000,C 0.000} C_DIS
LIN {X 274.235,Y 94.314,Z 220.061,A -161.021,B 90.000,C 0.000} C_DIS
LIN {X 273.657,Y 95.979,Z 221.628,A -160.673,B 90.000,C 0.000} C_DIS
LIN {X 273.643,Y 96.017,Z 221.742,A -160.665,B 90.000,C 0.000} C_DIS
LIN {X 273.241,Y 97.155,Z 222.780,A -160.426,B 90.000,C 0.000} C_DIS
LIN {X 273.167,Y 97.365,Z 222.937,A -160.382,B 90.000,C 0.000} C_DIS
LIN {X 273.148,Y 97.417,Z 223.022,A -160.372,B 90.000,C 0.000} C_DIS
LIN {X 273.119,Y 97.499,Z 223.108,A -160.354,B 90.000,C 0.000} C_DIS
LIN {X 273.041,Y 97.717,Z 223.278,A -160.308,B 90.000,C 0.000} C_DIS
LIN {X 272.987,Y 97.868,Z 223.449,A -160.277,B 90.000,C 0.000} C_DIS
LIN {X 272.720,Y 98.609,Z 224.018,A -160.121,B 90.000,C 0.000} C_DIS
LIN {X 272.710,Y 98.637,Z 224.132,A -160.115,B 90.000,C 0.000} C_DIS
LIN {X 272.577,Y 99.004,Z 224.359,A -160.038,B 90.000,C 0.000} C_DIS
LIN {X 272.522,Y 99.156,Z 224.530,A -160.006,B 90.000,C 0.000} C_DIS
LIN {X 272.219,Y 99.985,Z 225.158,A -159.832,B 90.000,C 0.000} C_DIS
LIN {X 272.186,Y 100.074,Z 225.253,A -159.813,B 90.000,C 0.000} C_DIS
LIN {X 271.958,Y 100.692,Z 225.739,A -159.683,B 90.000,C 0.000} C_DIS
LIN {X 271.889,Y 100.877,Z 225.839,A -159.644,B 90.000,C 0.000} C_DIS
LIN {X 271.824,Y 101.053,Z 226.010,A -159.607,B 90.000,C 0.000} C_DIS
LIN {X 271.457,Y 102.036,Z 226.749,A -159.400,B 90.000,C 0.000} C_DIS
LIN {X 271.165,Y 102.809,Z 227.267,A -159.236,B 90.000,C 0.000} C_DIS
LIN {X 271.076,Y 103.044,Z 227.397,A -159.187,B 90.000,C 0.000} C_DIS
LIN {X 270.308,Y 105.041,Z 228.690,A -158.764,B 90.000,C 0.000} C_DIS
LIN {X 269.693,Y 106.609,Z 229.594,A -158.431,B 90.000,C 0.000} C_DIS
LIN {X 269.590,Y 106.870,Z 229.629,A -158.376,B 90.000,C 0.000} C_DIS
LIN {X 269.559,Y 106.947,Z 229.486,A -158.359,B 90.000,C 0.000} C_DIS
LIN {X 269.122,Y 108.042,Z 227.281,A -158.126,B 90.000,C 0.000} C_DIS
LIN {X 268.901,Y 108.592,Z 226.180,A -158.009,B 90.000,C 0.000} C_DIS
LIN {X 268.886,Y 108.630,Z 226.066,A -158.001,B 90.000,C 0.000} C_DIS
LIN {X 268.458,Y 109.683,Z 223.840,A -157.777,B 90.000,C 0.000} C_DIS
LIN {X 268.029,Y 110.727,Z 221.609,A -157.554,B 90.000,C 0.000} C_DIS
LIN {X 267.607,Y 111.743,Z 219.364,A -157.336,B 90.000,C 0.000} C_DIS
LIN {X 267.189,Y 112.738,Z 217.109,A -157.123,B 90.000,C 0.000} C_DIS
LIN {X 266.777,Y 113.709,Z 214.843,A -156.915,B 90.000,C 0.000} C_DIS
LIN {X 266.368,Y 114.664,Z 212.569,A -156.709,B 90.000,C 0.000} C_DIS
LIN {X 265.963,Y 115.602,Z 210.287,A -156.508,B 90.000,C 0.000} C_DIS
LIN {X 265.564,Y 116.516,Z 207.995,A -156.311,B 90.000,C 0.000} C_DIS
LIN {X 265.170,Y 117.408,Z 205.693,A -156.118,B 90.000,C 0.000} C_DIS
LIN {X 264.783,Y 118.279,Z 203.382,A -155.930,B 90.000,C 0.000} C_DIS
LIN {X 264.407,Y 119.118,Z 201.057,A -155.748,B 90.000,C 0.000} C_DIS
LIN {X 264.034,Y 119.941,Z 198.726,A -155.569,B 90.000,C 0.000} C_DIS
LIN {X 263.674,Y 120.732,Z 196.382,A -155.398,B 90.000,C 0.000} C_DIS
LIN {X 263.322,Y 121.497,Z 194.028,A -155.231,B 90.000,C 0.000} C_DIS
LIN {X 262.984,Y 122.228,Z 191.662,A -155.072,B 90.000,C 0.000} C_DIS
LIN {X 262.655,Y 122.932,Z 189.286,A -154.919,B 90.000,C 0.000} C_DIS
LIN {X 262.594,Y 123.063,Z 188.857,A -154.890,B 90.000,C 0.000} C_DIS
LIN {X 262.589,Y 123.073,Z 188.784,A -154.888,B 90.000,C 0.000} C_DIS
LIN {X 262.300,Y 123.686,Z 186.378,A -154.754,B 90.000,C 0.000} C_DIS
LIN {X 262.014,Y 124.292,Z 183.969,A -154.622,B 90.000,C 0.000} C_DIS
LIN {X 261.750,Y 124.846,Z 181.546,A -154.500,B 90.000,C 0.000} C_DIS
LIN {X 261.491,Y 125.389,Z 179.119,A -154.382,B 90.000,C 0.000} C_DIS
LIN {X 261.280,Y 125.829,Z 176.668,A -154.285,B 90.000,C 0.000} C_DIS
LIN {X 261.097,Y 126.208,Z 174.203,A -154.202,B 90.000,C 0.000} C_DIS
LIN {X 261.001,Y 126.406,Z 172.680,A -154.159,B 90.000,C 0.000} C_DIS
LIN {X 260.699,Y 127.028,Z 175.082,A -154.022,B 90.000,C 0.000} C_DIS
LIN {X 260.678,Y 127.070,Z 175.258,A -154.013,B 90.000,C 0.000} C_DIS
LIN {X 260.668,Y 127.091,Z 175.443,A -154.008,B 90.000,C 0.000} C_DIS
LIN {X 260.648,Y 127.131,Z 175.543,A -153.999,B 90.000,C 0.000} C_DIS
LIN {X 260.511,Y 127.412,Z 176.567,A -153.938,B 90.000,C 0.000} C_DIS
LIN {X 260.496,Y 127.443,Z 176.806,A -153.931,B 90.000,C 0.000} C_DIS
LIN {X 260.198,Y 128.050,Z 179.115,A -153.797,B 90.000,C 0.000} C_DIS
LIN {X 260.188,Y 128.071,Z 179.244,A -153.792,B 90.000,C 0.000} C_DIS
LIN {X 260.152,Y 128.145,Z 179.466,A -153.776,B 90.000,C 0.000} C_DIS
LIN {X 260.141,Y 128.166,Z 179.594,A -153.772,B 90.000,C 0.000} C_DIS
LIN {X 259.890,Y 128.674,Z 181.403,A -153.660,B 90.000,C 0.000} C_DIS
LIN {X 259.860,Y 128.735,Z 181.801,A -153.646,B 90.000,C 0.000} C_DIS
LIN {X 259.844,Y 128.768,Z 181.915,A -153.639,B 90.000,C 0.000} C_DIS
LIN {X 259.830,Y 128.797,Z 181.972,A -153.633,B 90.000,C 0.000} C_DIS
LIN {X 259.824,Y 128.808,Z 182.029,A -153.630,B 90.000,C 0.000} C_DIS
LIN {X 259.588,Y 129.283,Z 183.707,A -153.525,B 90.000,C 0.000} C_DIS
LIN {X 259.577,Y 129.304,Z 183.864,A -153.521,B 90.000,C 0.000} C_DIS
LIN {X 259.564,Y 129.330,Z 183.963,A -153.515,B 90.000,C 0.000} C_DIS
LIN {X 259.518,Y 129.423,Z 184.177,A -153.494,B 90.000,C 0.000} C_DIS
LIN {X 259.392,Y 129.675,Z 185.123,A -153.439,B 90.000,C 0.000} C_DIS
LIN {X 259.382,Y 129.696,Z 185.286,A -153.434,B 90.000,C 0.000} C_DIS
LIN {X 259.358,Y 129.744,Z 185.386,A -153.423,B 90.000,C 0.000} C_DIS
LIN {X 259.343,Y 129.773,Z 185.423,A -153.417,B 90.000,C 0.000} C_DIS
LIN {X 259.334,Y 129.792,Z 185.531,A -153.413,B 90.000,C 0.000} C_DIS
LIN {X 259.124,Y 130.210,Z 186.922,A -153.320,B 90.000,C 0.000} C_DIS
LIN {X 258.879,Y 130.697,Z 188.742,A -153.213,B 90.000,C 0.000} C_DIS
LIN {X 258.539,Y 131.368,Z 190.848,A -153.064,B 90.000,C 0.000} C_DIS
LIN {X 258.522,Y 131.401,Z 191.075,A -153.057,B 90.000,C 0.000} C_DIS
LIN {X 258.356,Y 131.727,Z 191.986,A -152.985,B 90.000,C 0.000} C_DIS
LIN {X 258.326,Y 131.787,Z 192.346,A -152.971,B 90.000,C 0.000} C_DIS
LIN {X 258.310,Y 131.819,Z 192.384,A -152.964,B 90.000,C 0.000} C_DIS
LIN {X 258.290,Y 131.857,Z 192.498,A -152.956,B 90.000,C 0.000} C_DIS
LIN {X 258.283,Y 131.871,Z 192.611,A -152.952,B 90.000,C 0.000} C_DIS
LIN {X 258.179,Y 132.075,Z 193.180,A -152.907,B 90.000,C 0.000} C_DIS
LIN {X 258.171,Y 132.089,Z 193.294,A -152.904,B 90.000,C 0.000} C_DIS
LIN {X 258.154,Y 132.122,Z 193.408,A -152.897,B 90.000,C 0.000} C_DIS
LIN {X 258.140,Y 132.150,Z 193.465,A -152.891,B 90.000,C 0.000} C_DIS
LIN {X 258.134,Y 132.162,Z 193.522,A -152.888,B 90.000,C 0.000} C_DIS
LIN {X 257.980,Y 132.463,Z 194.356,A -152.821,B 90.000,C 0.000} C_DIS
LIN {X 257.975,Y 132.473,Z 194.455,A -152.819,B 90.000,C 0.000} C_DIS
LIN {X 257.839,Y 132.737,Z 195.229,A -152.760,B 90.000,C 0.000} C_DIS
LIN {X 257.834,Y 132.747,Z 195.342,A -152.758,B 90.000,C 0.000} C_DIS
LIN {X 257.799,Y 132.815,Z 195.542,A -152.743,B 90.000,C 0.000} C_DIS
LIN {X 257.793,Y 132.826,Z 195.627,A -152.741,B 90.000,C 0.000} C_DIS
LIN {X 257.655,Y 133.093,Z 196.400,A -152.681,B 90.000,C 0.000} C_DIS
LIN {X 257.650,Y 133.103,Z 196.500,A -152.679,B 90.000,C 0.000} C_DIS
LIN {X 257.529,Y 133.337,Z 197.076,A -152.627,B 90.000,C 0.000} C_DIS
LIN {X 257.435,Y 133.518,Z 197.632,A -152.587,B 90.000,C 0.000} C_DIS
LIN {X 257.056,Y 134.247,Z 199.808,A -152.424,B 90.000,C 0.000} C_DIS
LIN {X 256.932,Y 134.483,Z 200.387,A -152.372,B 90.000,C 0.000} C_DIS
